   LIN {X -3.618, Y 42.239, Z 30.600} C_DIS
   LIN {X -4.278, Y 41.274, Z 30.600} C_DIS
   LIN {X -4.651, Y 40.757, Z 30.600} C_DIS
   LIN {X -4.747, Y 40.345, Z 30.600} C_DIS
   LIN {X -4.925, Y 39.487, Z 30.600} C_DIS
   LIN {X -4.816, Y 38.644, Z 30.600} C_DIS
   LIN {X -4.756, Y 38.144, Z 30.600} C_DIS
   LIN {X -4.582, Y 37.523, Z 30.600} C_DIS
   LIN {X -4.417, Y 36.940, Z 30.600} C_DIS
   LIN {X -4.292, Y 36.475, Z 30.600} C_DIS
   LIN {X -4.004, Y 35.393, Z 30.600} C_DIS
   LIN {X -3.515, Y 33.337, Z 30.600} C_DIS
   LIN {X -3.455, Y 33.086, Z 30.600} C_DIS
   LIN {X -3.401, Y 32.820, Z 30.600} C_DIS
   LIN {X -2.886, Y 30.247, Z 30.600} C_DIS
   LIN {X -2.481, Y 27.620, Z 30.600} C_DIS
   LIN {X -2.317, Y 26.540, Z 30.600} C_DIS
   LIN {X -2.260, Y 25.886, Z 30.600} C_DIS
   LIN {X -1.842, Y 21.391, Z 30.600} C_DIS
   LIN {X -1.832, Y 19.498, Z 30.600} C_DIS
   LIN {X -1.874, Y 12.631, Z 30.600} C_DIS
   LIN {X -2.420, Y 7.896, Z 30.600} C_DIS
   LIN {X -2.629, Y 5.941, Z 30.600} C_DIS
   LIN {X -2.726, Y 5.309, Z 30.600} C_DIS
   LIN {X -3.850, Y 0.233, Z 30.600} C_DIS
   LIN {X -4.314, Y -1.891, Z 30.600} C_DIS
   LIN {X -4.758, Y -3.318, Z 30.600} C_DIS
   LIN {X -5.741, Y -6.496, Z 30.600} C_DIS
   LIN {X -6.964, Y -9.707, Z 30.600} C_DIS
   LIN {X -7.355, Y -10.723, Z 30.600} C_DIS
   LIN {X -7.726, Y -11.533, Z 30.600} C_DIS
   LIN {X -9.075, Y -14.528, Z 30.600} C_DIS
   LIN {X -10.538, Y -17.348, Z 30.600} C_DIS
   LIN {X -10.853, Y -17.945, Z 30.600} C_DIS
   LIN {X -11.124, Y -18.727, Z 30.600} C_DIS
   LIN {X -11.882, Y -20.944, Z 30.600} C_DIS
   LIN {X -11.789, Y -22.564, Z 30.600} C_DIS
   LIN {X -11.686, Y -24.649, Z 30.600} C_DIS
   LIN {X -10.821, Y -26.557, Z 30.600} C_DIS
   LIN {X -10.384, Y -27.445, Z 30.600} C_DIS
   LIN {X -8.989, Y -28.695, Z 30.600} C_DIS
   LIN {X -7.458, Y -30.118, Z 30.600} C_DIS
   LIN {X -6.898, Y -30.342, Z 30.600} C_DIS
   LIN {X -4.652, Y -31.135, Z 30.600} C_DIS
   LIN {X -2.453, Y -31.231, Z 30.600} C_DIS
   LIN {X -2.161, Y -31.241, Z 30.600} C_DIS
   LIN {X -1.901, Y -31.152, Z 30.600}
   LaserEnd_Ext()
   LIN {X -6.660, Y -29.360, Z 30.600}
   LaserStart_Ext()
   LIN {X 0.314, Y -29.360, Z 30.600}
   LaserEnd_Ext()
   LIN {X 1.927, Y -28.360, Z 30.600}
   LaserStart_Ext()
   LIN {X -7.880, Y -28.360, Z 30.600}
   LaserEnd_Ext()
   LIN {X -8.980, Y -27.360, Z 30.600}
   LaserStart_Ext()
   LIN {X -6.021, Y -27.360, Z 30.600}
   LaserEnd_Ext()
   LIN {X 0.049, Y -27.360, Z 30.600}
   LaserStart_Ext()
   LIN {X 2.964, Y -27.360, Z 30.600}
   LaserEnd_Ext()
   LIN {X 3.806, Y -26.360, Z 30.600}
   LaserStart_Ext()
   LIN {X 1.372, Y -26.360, Z 30.600}
   LaserEnd_Ext()
   LIN {X -7.389, Y -26.360, Z 30.600}
   LaserStart_Ext()
   LIN {X -9.804, Y -26.360, Z 30.600}
   LaserEnd_Ext()
   LIN {X -10.266, Y -25.360, Z 30.600}
   LaserStart_Ext()
   LIN {X -8.010, Y -25.360, Z 30.600}
   LaserEnd_Ext()
   LIN {X 2.006, Y -25.360, Z 30.600}
   LaserStart_Ext()
   LIN {X 4.260, Y -25.360, Z 30.600}
   LaserEnd_Ext()
   LIN {X 4.715, Y -24.360, Z 30.600}
   LaserStart_Ext()
   LIN {X 2.517, Y -24.360, Z 30.600}
   LaserEnd_Ext()
   LIN {X -8.601, Y -24.360, Z 30.600}
   LaserStart_Ext()
   LIN {X -10.699, Y -24.360, Z 30.600}
   LaserEnd_Ext()
   LIN {X -10.748, Y -23.360, Z 30.600}
   LaserStart_Ext()
   LIN {X -8.789, Y -23.360, Z 30.600}
   LaserEnd_Ext()
   LIN {X 2.910, Y -23.360, Z 30.600}
   LaserStart_Ext()
   LIN {X 4.998, Y -23.360, Z 30.600}
   LaserEnd_Ext()
   LIN {X 5.242, Y -22.360, Z 30.600}
   LaserStart_Ext()
   LIN {X 2.915, Y -22.360, Z 30.600}
   LaserEnd_Ext()
   LIN {X -8.897, Y -22.360, Z 30.600}
   LaserStart_Ext()
   LIN {X -10.799, Y -22.360, Z 30.600}
   LaserEnd_Ext()
   LIN {X -10.856, Y -21.360, Z 30.600}
   LaserStart_Ext()
   LIN {X -8.848, Y -21.360, Z 30.600}
   LaserEnd_Ext()
   LIN {X 2.920, Y -21.360, Z 30.600}
   LaserStart_Ext()
   LIN {X 5.487, Y -21.360, Z 30.600}
   LaserEnd_Ext()
   LIN {X 5.712, Y -20.360, Z 30.600}
   LaserStart_Ext()
   LIN {X 2.625, Y -20.360, Z 30.600}
   LaserEnd_Ext()
   LIN {X -8.405, Y -20.360, Z 30.600}
   LaserStart_Ext()
   LIN {X -10.626, Y -20.360, Z 30.600}
   LaserEnd_Ext()
   LIN {X -10.284, Y -19.360, Z 30.600}
   LaserStart_Ext()
   LIN {X -7.968, Y -19.360, Z 30.600}
   LaserEnd_Ext()
   LIN {X 2.112, Y -19.360, Z 30.600}
   LaserStart_Ext()
   LIN {X 5.927, Y -19.360, Z 30.600}
   LaserEnd_Ext()
   LIN {X 6.139, Y -18.360, Z 30.600}
   LaserStart_Ext()
   LIN {X 1.590, Y -18.360, Z 30.600}
   LaserEnd_Ext()
   LIN {X -7.498, Y -18.360, Z 30.600}
   LaserStart_Ext()
   LIN {X -9.938, Y -18.360, Z 30.600}
   LaserEnd_Ext()
   LIN {X -9.418, Y -17.360, Z 30.600}
   LaserStart_Ext()
   LIN {X -6.233, Y -17.360, Z 30.600}
   LaserEnd_Ext()
   LIN {X 0.313, Y -17.360, Z 30.600}
   LaserStart_Ext()
   LIN {X 6.327, Y -17.360, Z 30.600}
   LaserEnd_Ext()
   LIN {X 6.509, Y -16.360, Z 30.600}
   LaserStart_Ext()
   LIN {X -2.524, Y -16.360, Z 30.600}
   LaserEnd_Ext()
   LIN {X -3.563, Y -16.360, Z 30.600}
   LaserStart_Ext()
   LIN {X -8.899, Y -16.360, Z 30.600}
   LaserEnd_Ext()
   LIN {X -8.380, Y -15.360, Z 30.600}
   LaserStart_Ext()
   LIN {X 6.691, Y -15.360, Z 30.600}
   LaserEnd_Ext()
   LIN {X 6.872, Y -14.360, Z 30.600}
   LaserStart_Ext()
   LIN {X -7.902, Y -14.360, Z 30.600}
   LaserEnd_Ext()
   LIN {X -7.452, Y -13.360, Z 30.600}
   LaserStart_Ext()
   LIN {X 7.014, Y -13.360, Z 30.600}
   LaserEnd_Ext()
   LIN {X 7.155, Y -12.360, Z 30.600}
   LaserStart_Ext()
   LIN {X -7.001, Y -12.360, Z 30.600}
   LaserEnd_Ext()
   LIN {X -6.547, Y -11.360, Z 30.600}
   LaserStart_Ext()
   LIN {X 7.297, Y -11.360, Z 30.600}
   LaserEnd_Ext()
   LIN {X 7.438, Y -10.360, Z 30.600}
   LaserStart_Ext()
   LIN {X -6.143, Y -10.360, Z 30.600}
   LaserEnd_Ext()
   LIN {X -5.761, Y -9.360, Z 30.600}
   LaserStart_Ext()
   LIN {X 7.568, Y -9.360, Z 30.600}
   LaserEnd_Ext()
   LIN {X 7.662, Y -8.360, Z 30.600}
   LaserStart_Ext()
   LIN {X -5.381, Y -8.360, Z 30.600}
   LaserEnd_Ext()
   LIN {X -5.000, Y -7.360, Z 30.600}
   LaserStart_Ext()
   LIN {X 7.756, Y -7.360, Z 30.600}
   LaserEnd_Ext()
   LIN {X 7.850, Y -6.360, Z 30.600}
   LaserStart_Ext()
   LIN {X -4.652, Y -6.360, Z 30.600}
   LaserEnd_Ext()
   LIN {X -4.343, Y -5.360, Z 30.600}
   LaserStart_Ext()
   LIN {X 7.941, Y -5.360, Z 30.600}
   LaserEnd_Ext()
   LIN {X 8.031, Y -4.360, Z 30.600}
   LaserStart_Ext()
   LIN {X -4.033, Y -4.360, Z 30.600}
   LaserEnd_Ext()
   LIN {X -3.723, Y -3.360, Z 30.600}
   LaserStart_Ext()
   LIN {X 8.100, Y -3.360, Z 30.600}
   LaserEnd_Ext()
   LIN {X 8.152, Y -2.360, Z 30.600}
   LaserStart_Ext()
   LIN {X -3.412, Y -2.360, Z 30.600}
   LaserEnd_Ext()
   LIN {X -3.174, Y -1.360, Z 30.600}
   LaserStart_Ext()
   LIN {X 8.186, Y -1.360, Z 30.600}
   LaserEnd_Ext()
   LIN {X 8.211, Y -0.360, Z 30.600}
   LaserStart_Ext()
   LIN {X -2.956, Y -0.360, Z 30.600}
   LaserEnd_Ext()
   LIN {X -2.735, Y 0.640, Z 30.600}
   LaserStart_Ext()
   LIN {X 8.237, Y 0.640, Z 30.600}
   LaserEnd_Ext()
   LIN {X 8.262, Y 1.640, Z 30.600}
   LaserStart_Ext()
   LIN {X -2.514, Y 1.640, Z 30.600}
   LaserEnd_Ext()
   LIN {X -2.293, Y 2.640, Z 30.600}
   LaserStart_Ext()
   LIN {X 8.288, Y 2.640, Z 30.600}
   LaserEnd_Ext()
   LIN {X 8.271, Y 3.640, Z 30.600}
   LaserStart_Ext()
   LIN {X -2.071, Y 3.640, Z 30.600}
   LaserEnd_Ext()
   LIN {X -1.850, Y 4.640, Z 30.600}
   LaserStart_Ext()
   LIN {X 8.247, Y 4.640, Z 30.600}
   LaserEnd_Ext()
   LIN {X 8.223, Y 5.640, Z 30.600}
   LaserStart_Ext()
   LIN {X -1.664, Y 5.640, Z 30.600}
   LaserEnd_Ext()
   LIN {X -1.549, Y 6.640, Z 30.600}
   LaserStart_Ext()
   LIN {X 8.199, Y 6.640, Z 30.600}
   LaserEnd_Ext()
   LIN {X 8.175, Y 7.640, Z 30.600}
   LaserStart_Ext()
   LIN {X -1.441, Y 7.640, Z 30.600}
   LaserEnd_Ext()
   LIN {X -1.327, Y 8.640, Z 30.600}
   LaserStart_Ext()
   LIN {X 8.137, Y 8.640, Z 30.600}
   LaserEnd_Ext()
   LIN {X 8.089, Y 9.640, Z 30.600}
   LaserStart_Ext()
   LIN {X -1.212, Y 9.640, Z 30.600}
   LaserEnd_Ext()
   LIN {X -1.097, Y 10.640, Z 30.600}
   LaserStart_Ext()
   LIN {X 8.042, Y 10.640, Z 30.600}
   LaserEnd_Ext()
   LIN {X 7.995, Y 11.640, Z 30.600}
   LaserStart_Ext()
   LIN {X -0.982, Y 11.640, Z 30.600}
   LaserEnd_Ext()
   LIN {X -0.874, Y 12.640, Z 30.600}
   LaserStart_Ext()
   LIN {X 7.910, Y 12.640, Z 30.600}
   LaserEnd_Ext()
   LIN {X 7.806, Y 13.640, Z 30.600}
   LaserStart_Ext()
   LIN {X -0.868, Y 13.640, Z 30.600}
   LaserEnd_Ext()
   LIN {X -0.862, Y 14.640, Z 30.600}
   LaserStart_Ext()
   LIN {X 7.702, Y 14.640, Z 30.600}
   LaserEnd_Ext()
   LIN {X 7.569, Y 15.640, Z 30.600}
   LaserStart_Ext()
   LIN {X -0.856, Y 15.640, Z 30.600}
   LaserEnd_Ext()
   LIN {X -0.850, Y 16.640, Z 30.600}
   LaserStart_Ext()
   LIN {X 7.431, Y 16.640, Z 30.600}
   LaserEnd_Ext()
   LIN {X 7.292, Y 17.640, Z 30.600}
   LaserStart_Ext()
   LIN {X -0.844, Y 17.640, Z 30.600}
   LaserEnd_Ext()
   LIN {X -0.838, Y 18.640, Z 30.600}
   LaserStart_Ext()
   LIN {X 7.154, Y 18.640, Z 30.600}
   LaserEnd_Ext()
   LIN {X 7.015, Y 19.640, Z 30.600}
   LaserStart_Ext()
   LIN {X -0.833, Y 19.640, Z 30.600}
   LaserEnd_Ext()
   LIN {X -0.838, Y 20.640, Z 30.600}
   LaserStart_Ext()
   LIN {X 6.864, Y 20.640, Z 30.600}
   LaserEnd_Ext()
   LIN {X 6.713, Y 21.640, Z 30.600}
   LaserStart_Ext()
   LIN {X -0.861, Y 21.640, Z 30.600}
   LaserEnd_Ext()
   LIN {X -0.954, Y 22.640, Z 30.600}
   LaserStart_Ext()
   LIN {X 6.561, Y 22.640, Z 30.600}
   LaserEnd_Ext()
   LIN {X 6.391, Y 23.640, Z 30.600}
   LaserStart_Ext()
   LIN {X -1.047, Y 23.640, Z 30.600}
   LaserEnd_Ext()
   LIN {X -1.139, Y 24.640, Z 30.600}
   LaserStart_Ext()
   LIN {X 6.173, Y 24.640, Z 30.600}
   LaserEnd_Ext()
   LIN {X 5.937, Y 25.640, Z 30.600}
   LaserStart_Ext()
   LIN {X -1.232, Y 25.640, Z 30.600}
   LaserEnd_Ext()
   LIN {X -1.323, Y 26.640, Z 30.600}
   LaserStart_Ext()
   LIN {X 5.697, Y 26.640, Z 30.600}
   LaserEnd_Ext()
   LIN {X 5.476, Y 27.640, Z 30.600}
   LaserStart_Ext()
   LIN {X -1.473, Y 27.640, Z 30.600}
   LaserEnd_Ext()
   LIN {X -1.627, Y 28.640, Z 30.600}
   LaserStart_Ext()
   LIN {X 5.270, Y 28.640, Z 30.600}
   LaserEnd_Ext()
   LIN {X 5.064, Y 29.640, Z 30.600}
   LaserStart_Ext()
   LIN {X -1.781, Y 29.640, Z 30.600}
   LaserEnd_Ext()
   LIN {X -1.945, Y 30.640, Z 30.600}
   LaserStart_Ext()
   LIN {X 4.824, Y 30.640, Z 30.600}
   LaserEnd_Ext()
   LIN {X 4.555, Y 31.640, Z 30.600}
   LaserStart_Ext()
   LIN {X -2.145, Y 31.640, Z 30.600}
   LaserEnd_Ext()
   LIN {X -2.345, Y 32.640, Z 30.600}
   LaserStart_Ext()
   LIN {X 4.287, Y 32.640, Z 30.600}
   LaserEnd_Ext()
   LIN {X 4.007, Y 33.640, Z 30.600}
   LaserStart_Ext()
   LIN {X -2.559, Y 33.640, Z 30.600}
   LaserEnd_Ext()
   LIN {X -2.797, Y 34.640, Z 30.600}
   LaserStart_Ext()
   LIN {X 3.712, Y 34.640, Z 30.600}
   LaserEnd_Ext()
   LIN {X 3.413, Y 35.640, Z 30.600}
   LaserStart_Ext()
   LIN {X -3.035, Y 35.640, Z 30.600}
   LaserEnd_Ext()
   LIN {X -3.301, Y 36.640, Z 30.600}
   LaserStart_Ext()
   LIN {X 3.097, Y 36.640, Z 30.600}
   LaserEnd_Ext()
   LIN {X 2.773, Y 37.640, Z 30.600}
   LaserStart_Ext()
   LIN {X -3.576, Y 37.640, Z 30.600}
   LaserEnd_Ext()
   LIN {X -3.808, Y 38.640, Z 30.600}
   LaserStart_Ext()
   LIN {X 2.438, Y 38.640, Z 30.600}
   LaserEnd_Ext()
   LIN {X 2.090, Y 39.640, Z 30.600}
   LaserStart_Ext()
   LIN {X -3.872, Y 39.640, Z 30.600}
   LaserEnd_Ext()
   LIN {X -3.502, Y 40.640, Z 30.600}
   LaserStart_Ext()
   LIN {X 1.632, Y 40.640, Z 30.600}
   LaserEnd_Ext()
   LIN {X 0.709, Y 41.640, Z 30.600}
   LaserStart_Ext()
   LIN {X -2.425, Y 41.640, Z 30.600}
   LaserEnd_Ext()
   LIN {X -5.717, Y -18.241, Z 31.450}
   LaserStart_Ext()
   LIN {X -5.008, Y -17.700, Z 31.450} C_DIS
   LIN {X -3.784, Y -17.409, Z 31.450} C_DIS
   LIN {X -3.008, Y -17.226, Z 31.450} C_DIS
   LIN {X -2.409, Y -17.339, Z 31.450} C_DIS
   LIN {X -0.901, Y -17.619, Z 31.450} C_DIS
   LIN {X 0.539, Y -18.651, Z 31.450} C_DIS
   LIN {X 0.826, Y -18.857, Z 31.450} C_DIS
   LIN {X 1.021, Y -19.237, Z 31.450} C_DIS
   LIN {X 1.994, Y -21.116, Z 31.450} C_DIS
   LIN {X 1.991, Y -22.729, Z 31.450} C_DIS
   LIN {X 1.988, Y -23.292, Z 31.450} C_DIS
   LIN {X 1.755, Y -23.747, Z 31.450} C_DIS
   LIN {X 0.880, Y -25.483, Z 31.450} C_DIS
   LIN {X -0.658, Y -26.657, Z 31.450} C_DIS
   LIN {X -0.782, Y -26.750, Z 31.450} C_DIS
   LIN {X -1.016, Y -26.803, Z 31.450} C_DIS
   LIN {X -2.872, Y -27.227, Z 31.450} C_DIS
   LIN {X -4.055, Y -26.995, Z 31.450} C_DIS
   LIN {X -4.899, Y -26.827, Z 31.450} C_DIS
   LIN {X -5.838, Y -26.159, Z 31.450} C_DIS
   LIN {X -6.583, Y -25.632, Z 31.450} C_DIS
   LIN {X -6.989, Y -24.951, Z 31.450} C_DIS
   LIN {X -7.647, Y -23.841, Z 31.450} C_DIS
   LIN {X -7.782, Y -22.606, Z 31.450} C_DIS
   LIN {X -7.876, Y -21.767, Z 31.450} C_DIS
   LIN {X -7.421, Y -20.706, Z 31.450} C_DIS
   LIN {X -6.650, Y -18.943, Z 31.450} C_DIS
   LIN {X -5.717, Y -18.241, Z 31.450}
   LaserEnd_Ext()
   LIN {X -7.202, Y -30.145, Z 31.450}
   LaserStart_Ext()
   LIN {X -7.333, Y -30.100, Z 31.450} C_DIS
   LIN {X -7.451, Y -30.002, Z 31.450} C_DIS
   LIN {X -10.203, Y -27.537, Z 31.450} C_DIS
   LIN {X -11.201, Y -25.513, Z 31.450} C_DIS
   LIN {X -11.604, Y -24.623, Z 31.450} C_DIS
   LIN {X -11.652, Y -23.650, Z 31.450} C_DIS
   LIN {X -11.809, Y -20.918, Z 31.450} C_DIS
   LIN {X -10.940, Y -18.374, Z 31.450} C_DIS
   LIN {X -10.787, Y -17.916, Z 31.450} C_DIS
   LIN {X -10.416, Y -17.192, Z 31.450} C_DIS
   LIN {X -9.022, Y -14.506, Z 31.450} C_DIS
   LIN {X -7.603, Y -11.355, Z 31.450} C_DIS
   LIN {X -7.335, Y -10.755, Z 31.450} C_DIS
   LIN {X -7.135, Y -10.224, Z 31.450} C_DIS
   LIN {X -5.720, Y -6.507, Z 31.450} C_DIS
   LIN {X -4.429, Y -2.333, Z 31.450} C_DIS
   LIN {X -4.342, Y -2.051, Z 31.450} C_DIS
   LIN {X -4.236, Y -1.572, Z 31.450} C_DIS
   LIN {X -2.754, Y 5.125, Z 31.450} C_DIS
   LIN {X -2.686, Y 5.572, Z 31.450} C_DIS
   LIN {X -2.537, Y 6.955, Z 31.450} C_DIS
   LIN {X -1.884, Y 12.627, Z 31.450} C_DIS
   LIN {X -1.848, Y 18.597, Z 31.450} C_DIS
   LIN {X -1.861, Y 21.319, Z 31.450} C_DIS
   LIN {X -2.299, Y 26.031, Z 31.450} C_DIS
   LIN {X -2.356, Y 26.579, Z 31.450} C_DIS
   LIN {X -2.912, Y 30.155, Z 31.450} C_DIS
   LIN {X -2.934, Y 30.294, Z 31.450} C_DIS
   LIN {X -2.965, Y 30.445, Z 31.450} C_DIS
   LIN {X -3.510, Y 33.132, Z 31.450} C_DIS
   LIN {X -3.950, Y 34.966, Z 31.450} C_DIS
   LIN {X -4.064, Y 35.438, Z 31.450} C_DIS
   LIN {X -4.163, Y 35.801, Z 31.450} C_DIS
   LIN {X -4.481, Y 36.983, Z 31.450} C_DIS
   LIN {X -4.646, Y 37.568, Z 31.450} C_DIS
   LIN {X -4.822, Y 38.187, Z 31.450} C_DIS
   LIN {X -4.952, Y 39.128, Z 31.450} C_DIS
   LIN {X -4.997, Y 39.480, Z 31.450} C_DIS
   LIN {X -4.933, Y 39.787, Z 31.450} C_DIS
   LIN {X -4.730, Y 40.786, Z 31.450} C_DIS
   LIN {X -3.916, Y 42.007, Z 31.450} C_DIS
   LIN {X -3.783, Y 42.202, Z 31.450} C_DIS
   LIN {X -3.444, Y 42.338, Z 31.450} C_DIS
   LIN {X -1.107, Y 43.314, Z 31.450} C_DIS
   LIN {X -0.169, Y 43.123, Z 31.450} C_DIS
   LIN {X 0.604, Y 42.964, Z 31.450} C_DIS
   LIN {X 1.747, Y 42.113, Z 31.450} C_DIS
   LIN {X 2.000, Y 41.925, Z 31.450} C_DIS
   LIN {X 2.087, Y 41.778, Z 31.450} C_DIS
   LIN {X 2.744, Y 40.655, Z 31.450} C_DIS
   LIN {X 3.191, Y 39.389, Z 31.450} C_DIS
   LIN {X 3.246, Y 39.232, Z 31.450} C_DIS
   LIN {X 3.477, Y 38.542, Z 31.450} C_DIS
   LIN {X 3.893, Y 37.300, Z 31.450} C_DIS
   LIN {X 4.023, Y 36.889, Z 31.450} C_DIS
   LIN {X 4.480, Y 35.439, Z 31.450} C_DIS
   LIN {X 4.741, Y 34.561, Z 31.450} C_DIS
   LIN {X 5.244, Y 32.823, Z 31.450} C_DIS
   LIN {X 5.775, Y 30.842, Z 31.450} C_DIS
   LIN {X 6.172, Y 28.912, Z 31.450} C_DIS
   LIN {X 6.972, Y 25.578, Z 31.450} C_DIS
   LIN {X 7.445, Y 23.404, Z 31.450} C_DIS
   LIN {X 8.277, Y 17.909, Z 31.450} C_DIS
   LIN {X 8.637, Y 15.308, Z 31.450} C_DIS
   LIN {X 8.987, Y 11.946, Z 31.450} C_DIS
   LIN {X 9.209, Y 7.250, Z 31.450} C_DIS
   LIN {X 9.310, Y 3.065, Z 31.450} C_DIS
   LIN {X 9.164, Y -2.691, Z 31.450} C_DIS
   LIN {X 9.094, Y -4.040, Z 31.450} C_DIS
   LIN {X 8.728, Y -8.094, Z 31.450} C_DIS
   LIN {X 8.571, Y -9.762, Z 31.450} C_DIS
   LIN {X 8.269, Y -11.897, Z 31.450} C_DIS
   LIN {X 7.918, Y -14.449, Z 31.450} C_DIS
   LIN {X 7.636, Y -16.049, Z 31.450} C_DIS
   LIN {X 7.235, Y -18.253, Z 31.450} C_DIS
   LIN {X 6.652, Y -21.011, Z 31.450} C_DIS
   LIN {X 6.600, Y -21.250, Z 31.450} C_DIS
   LIN {X 6.472, Y -21.773, Z 31.450} C_DIS
   LIN {X 5.835, Y -24.421, Z 31.450} C_DIS
   LIN {X 5.233, Y -25.767, Z 31.450} C_DIS
   LIN {X 4.574, Y -27.217, Z 31.450} C_DIS
   LIN {X 2.371, Y -29.339, Z 31.450} C_DIS
   LIN {X 1.831, Y -29.865, Z 31.450} C_DIS
   LIN {X 1.421, Y -30.017, Z 31.450} C_DIS
   LIN {X -1.962, Y -31.179, Z 31.450} C_DIS
   LIN {X -3.938, Y -31.107, Z 31.450} C_DIS
   LIN {X -4.513, Y -31.100, Z 31.450} C_DIS
   LIN {X -7.202, Y -30.145, Z 31.450}
   LaserEnd_Ext()
   LIN {X 7.602, Y -9.387, Z 31.450}
   LaserStart_Ext()
   LIN {X 7.602, Y 15.492, Z 31.450}
   LaserEnd_Ext()
   LIN {X 6.602, Y 22.292, Z 31.450}
   LaserStart_Ext()
   LIN {X 6.602, Y -16.145, Z 31.450}
   LaserEnd_Ext()
   LIN {X 5.602, Y -21.121, Z 31.450}
   LaserStart_Ext()
   LIN {X 5.602, Y 27.002, Z 31.450}
   LaserEnd_Ext()
   LIN {X 4.602, Y 31.355, Z 31.450}
   LaserStart_Ext()
   LIN {X 4.602, Y -24.728, Z 31.450}
   LaserEnd_Ext()
   LIN {X 3.602, Y -26.765, Z 31.450}
   LaserStart_Ext()
   LIN {X 3.602, Y 34.884, Z 31.450}
   LaserEnd_Ext()
   LIN {X 2.602, Y 38.005, Z 31.450}
   LaserStart_Ext()
   LIN {X 2.602, Y -20.115, Z 31.450}
   LaserEnd_Ext()
   LIN {X 2.602, Y -24.289, Z 31.450}
   LaserStart_Ext()
   LIN {X 2.602, Y -27.729, Z 31.450}
   LaserEnd_Ext()
   LIN {X 1.602, Y -28.693, Z 31.450}
   LaserStart_Ext()
   LIN {X 1.602, Y -26.174, Z 31.450}
   LaserEnd_Ext()
   LIN {X 1.602, Y -18.228, Z 31.450}
   LaserStart_Ext()
   LIN {X 1.602, Y 40.626, Z 31.450}
   LaserEnd_Ext()
   LIN {X 0.602, Y 41.719, Z 31.450}
   LaserStart_Ext()
   LIN {X 0.602, Y -17.466, Z 31.450}
   LaserEnd_Ext()
   LIN {X 0.602, Y -26.953, Z 31.450}
   LaserStart_Ext()
   LIN {X 0.602, Y -29.241, Z 31.450}
   LaserEnd_Ext()
   LIN {X -0.398, Y -29.585, Z 31.450}
   LaserStart_Ext()
   LIN {X -0.398, Y -27.672, Z 31.450}
   LaserEnd_Ext()
   LIN {X -0.398, Y -16.756, Z 31.450}
   LaserStart_Ext()
   LIN {X -0.398, Y 42.150, Z 31.450}
   LaserEnd_Ext()
   LIN {X -1.398, Y 42.109, Z 31.450}
   LaserStart_Ext()
   LIN {X -1.398, Y 26.928, Z 31.450}
   LaserEnd_Ext()
   LIN {X -1.398, Y 8.105, Z 31.450}
   LaserStart_Ext()
   LIN {X -1.398, Y -16.510, Z 31.450}
   LaserEnd_Ext()
   LIN {X -1.398, Y -27.916, Z 31.450}
   LaserStart_Ext()
   LIN {X -1.398, Y -29.928, Z 31.450}
   LaserEnd_Ext()
   LIN {X -2.398, Y -30.163, Z 31.450}
   LaserStart_Ext()
   LIN {X -2.398, Y -28.144, Z 31.450}
   LaserEnd_Ext()
   LIN {X -2.398, Y -16.323, Z 31.450}
   LaserStart_Ext()
   LIN {X -2.398, Y 2.106, Z 31.450}
   LaserEnd_Ext()
   LIN {X -2.398, Y 32.682, Z 31.450}
   LaserStart_Ext()
   LIN {X -2.398, Y 41.691, Z 31.450}
   LaserEnd_Ext()
   LIN {X -3.398, Y 40.982, Z 31.450}
   LaserStart_Ext()
   LIN {X -3.398, Y 36.808, Z 31.450}
   LaserEnd_Ext()
   LIN {X -3.398, Y -2.383, Z 31.450}
   LaserStart_Ext()
   LIN {X -3.398, Y -16.290, Z 31.450}
   LaserEnd_Ext()
   LIN {X -3.398, Y -28.143, Z 31.450}
   LaserStart_Ext()
   LIN {X -3.398, Y -30.126, Z 31.450}
   LaserEnd_Ext()
   LIN {X -4.398, Y -30.080, Z 31.450}
   LaserStart_Ext()
   LIN {X -4.398, Y -27.946, Z 31.450}
   LaserEnd_Ext()
   LIN {X -4.398, Y -16.527, Z 31.450}
   LaserStart_Ext()
   LIN {X -4.398, Y -5.618, Z 31.450}
   LaserEnd_Ext()
   LIN {X -5.398, Y -8.472, Z 31.450}
   LaserStart_Ext()
   LIN {X -5.398, Y -16.781, Z 31.450}
   LaserEnd_Ext()
   LIN {X -5.398, Y -27.694, Z 31.450}
   LaserStart_Ext()
   LIN {X -5.398, Y -29.724, Z 31.450}
   LaserEnd_Ext()
   LIN {X -6.398, Y -29.369, Z 31.450}
   LaserStart_Ext()
   LIN {X -6.398, Y -26.988, Z 31.450}
   LaserEnd_Ext()
   LIN {X -6.398, Y -17.502, Z 31.450}
   LaserStart_Ext()
   LIN {X -6.398, Y -11.105, Z 31.450}
   LaserEnd_Ext()
   LIN {X -7.398, Y -13.335, Z 31.450}
   LaserStart_Ext()
   LIN {X -7.398, Y -18.280, Z 31.450}
   LaserEnd_Ext()
   LIN {X -7.398, Y -26.209, Z 31.450}
   LaserStart_Ext()
   LIN {X -7.398, Y -28.707, Z 31.450}
   LaserEnd_Ext()
   LIN {X -8.398, Y -27.811, Z 31.450}
   LaserStart_Ext()
   LIN {X -8.398, Y -24.536, Z 31.450}
   LaserEnd_Ext()
   LIN {X -8.398, Y -20.448, Z 31.450}
   LaserStart_Ext()
   LIN {X -8.398, Y -15.474, Z 31.450}
   LaserEnd_Ext()
   LIN {X -9.398, Y -17.401, Z 31.450}
   LaserStart_Ext()
   LIN {X -9.398, Y -26.909, Z 31.450}
   LaserEnd_Ext()
   LIN {X -10.398, Y -24.862, Z 31.450}
   LaserStart_Ext()
   LIN {X -10.398, Y -19.882, Z 31.450}
   LaserEnd_Ext()
   LIN {X -2.796, Y -27.179, Z 32.300}
   LaserStart_Ext()
   LIN {X -4.245, Y -26.895, Z 32.300} C_DIS
   LIN {X -4.813, Y -26.785, Z 32.300} C_DIS
   LIN {X -5.177, Y -26.529, Z 32.300} C_DIS
   LIN {X -6.499, Y -25.593, Z 32.300} C_DIS
   LIN {X -7.463, Y -23.980, Z 32.300} C_DIS
   LIN {X -7.568, Y -23.805, Z 32.300} C_DIS
   LIN {X -7.590, Y -23.612, Z 32.300} C_DIS
   LIN {X -7.802, Y -21.731, Z 32.300} C_DIS
   LIN {X -6.614, Y -18.964, Z 32.300} C_DIS
   LIN {X -4.937, Y -17.655, Z 32.300} C_DIS
   LIN {X -2.934, Y -17.178, Z 32.300} C_DIS
   LIN {X -2.093, Y -17.333, Z 32.300} C_DIS
   LIN {X -0.836, Y -17.567, Z 32.300} C_DIS
   LIN {X 0.042, Y -18.196, Z 32.300} C_DIS
   LIN {X 0.893, Y -18.800, Z 32.300} C_DIS
   LIN {X 1.517, Y -19.995, Z 32.300} C_DIS
   LIN {X 2.067, Y -21.057, Z 32.300} C_DIS
   LIN {X 2.065, Y -22.216, Z 32.300} C_DIS
   LIN {X 2.066, Y -23.233, Z 32.300} C_DIS
   LIN {X 1.275, Y -24.812, Z 32.300} C_DIS
   LIN {X 0.967, Y -25.422, Z 32.300} C_DIS
   LIN {X 0.622, Y -25.686, Z 32.300} C_DIS
   LIN {X -0.683, Y -26.691, Z 32.300} C_DIS
   LIN {X -1.785, Y -26.948, Z 32.300} C_DIS
   LIN {X -2.796, Y -27.179, Z 32.300}
   LaserEnd_Ext()
   LIN {X 4.664, Y -27.150, Z 32.300}
   LaserStart_Ext()
   LIN {X 4.229, Y -27.568, Z 32.300} C_DIS
   LIN {X 1.936, Y -29.800, Z 32.300} C_DIS
   LIN {X 0.194, Y -30.445, Z 32.300} C_DIS
   LIN {X -1.762, Y -31.117, Z 32.300} C_DIS
   LIN {X -2.905, Y -31.075, Z 32.300} C_DIS
   LIN {X -4.408, Y -31.057, Z 32.300} C_DIS
   LIN {X -6.317, Y -30.380, Z 32.300} C_DIS
   LIN {X -7.237, Y -30.063, Z 32.300} C_DIS
   LIN {X -8.072, Y -29.376, Z 32.300} C_DIS
   LIN {X -10.023, Y -27.629, Z 32.300} C_DIS
   LIN {X -11.437, Y -24.759, Z 32.300} C_DIS
   LIN {X -11.523, Y -24.596, Z 32.300} C_DIS
   LIN {X -11.538, Y -24.342, Z 32.300} C_DIS
   LIN {X -11.736, Y -20.891, Z 32.300} C_DIS
   LIN {X -11.188, Y -19.289, Z 32.300} C_DIS
   LIN {X -10.721, Y -17.888, Z 32.300} C_DIS
   LIN {X -9.586, Y -15.672, Z 32.300} C_DIS
   LIN {X -8.969, Y -14.483, Z 32.300} C_DIS
   LIN {X -8.341, Y -13.089, Z 32.300} C_DIS
   LIN {X -7.327, Y -10.818, Z 32.300} C_DIS
   LIN {X -6.572, Y -8.810, Z 32.300} C_DIS
   LIN {X -5.699, Y -6.518, Z 32.300} C_DIS
   LIN {X -4.903, Y -3.945, Z 32.300} C_DIS
   LIN {X -4.340, Y -2.108, Z 32.300} C_DIS
   LIN {X -3.652, Y 1.011, Z 32.300} C_DIS
   LIN {X -2.782, Y 4.941, Z 32.300} C_DIS
   LIN {X -2.742, Y 5.203, Z 32.300} C_DIS
   LIN {X -2.655, Y 6.015, Z 32.300} C_DIS
   LIN {X -1.893, Y 12.624, Z 32.300} C_DIS
   LIN {X -1.863, Y 17.695, Z 32.300} C_DIS
   LIN {X -1.880, Y 21.247, Z 32.300} C_DIS
   LIN {X -2.251, Y 25.238, Z 32.300} C_DIS
   LIN {X -2.395, Y 26.628, Z 32.300} C_DIS
   LIN {X -2.982, Y 30.341, Z 32.300} C_DIS
   LIN {X -3.375, Y 32.263, Z 32.300} C_DIS
   LIN {X -3.564, Y 33.178, Z 32.300} C_DIS
   LIN {X -3.746, Y 33.923, Z 32.300} C_DIS
   LIN {X -4.124, Y 35.483, Z 32.300} C_DIS
   LIN {X -4.376, Y 36.413, Z 32.300} C_DIS
   LIN {X -4.544, Y 37.027, Z 32.300} C_DIS
   LIN {X -4.739, Y 37.706, Z 32.300} C_DIS
   LIN {X -4.889, Y 38.230, Z 32.300} C_DIS
   LIN {X -4.940, Y 38.602, Z 32.300} C_DIS
   LIN {X -5.067, Y 39.511, Z 32.300} C_DIS
   LIN {X -4.820, Y 40.724, Z 32.300} C_DIS
   LIN {X -4.793, Y 40.854, Z 32.300} C_DIS
   LIN {X -4.713, Y 40.975, Z 32.300} C_DIS
   LIN {X -3.866, Y 42.240, Z 32.300} C_DIS
   LIN {X -3.583, Y 42.458, Z 32.300} C_DIS
   LIN {X -2.040, Y 43.009, Z 32.300} C_DIS
   LIN {X -1.185, Y 43.365, Z 32.300} C_DIS
   LIN {X -0.330, Y 43.192, Z 32.300} C_DIS
   LIN {X 0.526, Y 43.020, Z 32.300} C_DIS
   LIN {X 1.009, Y 42.664, Z 32.300} C_DIS
   LIN {X 1.925, Y 41.984, Z 32.300} C_DIS
   LIN {X 2.653, Y 40.747, Z 32.300} C_DIS
   LIN {X 3.169, Y 39.316, Z 32.300} C_DIS
   LIN {X 3.621, Y 37.984, Z 32.300} C_DIS
   LIN {X 3.795, Y 37.465, Z 32.300} C_DIS
   LIN {X 4.490, Y 35.270, Z 32.300} C_DIS
   LIN {X 4.547, Y 35.089, Z 32.300} C_DIS
   LIN {X 4.579, Y 34.979, Z 32.300} C_DIS
   LIN {X 5.364, Y 32.263, Z 32.300} C_DIS
   LIN {X 5.599, Y 31.386, Z 32.300} C_DIS
   LIN {X 5.776, Y 30.532, Z 32.300} C_DIS
   LIN {X 6.829, Y 26.137, Z 32.300} C_DIS
   LIN {X 7.453, Y 23.272, Z 32.300} C_DIS
   LIN {X 8.549, Y 16.032, Z 32.300} C_DIS
   LIN {X 8.597, Y 15.682, Z 32.300} C_DIS
   LIN {X 8.998, Y 11.830, Z 32.300} C_DIS
   LIN {X 9.253, Y 6.448, Z 32.300} C_DIS
   LIN {X 9.328, Y 3.336, Z 32.300} C_DIS
   LIN {X 9.158, Y -3.325, Z 32.300} C_DIS
   LIN {X 9.119, Y -4.081, Z 32.300} C_DIS
   LIN {X 8.658, Y -9.193, Z 32.300} C_DIS
   LIN {X 8.606, Y -9.786, Z 32.300} C_DIS
   LIN {X 8.571, Y -10.054, Z 32.300} C_DIS
   LIN {X 7.972, Y -14.398, Z 32.300} C_DIS
   LIN {X 7.422, Y -17.520, Z 32.300} C_DIS
   LIN {X 7.302, Y -18.182, Z 32.300} C_DIS
   LIN {X 7.076, Y -19.252, Z 32.300} C_DIS
   LIN {X 6.674, Y -21.180, Z 32.300} C_DIS
   LIN {X 6.462, Y -22.087, Z 32.300} C_DIS
   LIN {X 5.916, Y -24.353, Z 32.300} C_DIS
   LIN {X 4.793, Y -26.864, Z 32.300} C_DIS
   LIN {X 4.664, Y -27.150, Z 32.300}
   LaserEnd_Ext()
   LIN {X -3.144, Y 41.522, Z 32.300}
   LaserStart_Ext()
   LIN {X 0.870, Y 41.522, Z 32.300}
   LaserEnd_Ext()
   LIN {X 1.625, Y 40.522, Z 32.300}
   LaserStart_Ext()
   LIN {X -3.812, Y 40.522, Z 32.300}
   LaserEnd_Ext()
   LIN {X -4.044, Y 39.522, Z 32.300}
   LaserStart_Ext()
   LIN {X 2.035, Y 39.522, Z 32.300}
   LaserEnd_Ext()
   LIN {X 2.383, Y 38.522, Z 32.300}
   LaserStart_Ext()
   LIN {X -3.919, Y 38.522, Z 32.300}
   LaserEnd_Ext()
   LIN {X -3.646, Y 37.522, Z 32.300}
   LaserStart_Ext()
   LIN {X 2.722, Y 37.522, Z 32.300}
   LaserEnd_Ext()
   LIN {X 3.045, Y 36.522, Z 32.300}
   LaserStart_Ext()
   LIN {X -3.370, Y 36.522, Z 32.300}
   LaserEnd_Ext()
   LIN {X -3.105, Y 35.522, Z 32.300}
   LaserStart_Ext()
   LIN {X 3.361, Y 35.522, Z 32.300}
   LaserEnd_Ext()
   LIN {X 3.670, Y 34.522, Z 32.300}
   LaserStart_Ext()
   LIN {X -2.862, Y 34.522, Z 32.300}
   LaserEnd_Ext()
   LIN {X -2.619, Y 33.522, Z 32.300}
   LaserStart_Ext()
   LIN {X 3.959, Y 33.522, Z 32.300}
   LaserEnd_Ext()
   LIN {X 4.249, Y 32.522, Z 32.300}
   LaserStart_Ext()
   LIN {X -2.407, Y 32.522, Z 32.300}
   LaserEnd_Ext()
   LIN {X -2.203, Y 31.522, Z 32.300}
   LaserStart_Ext()
   LIN {X 4.528, Y 31.522, Z 32.300}
   LaserEnd_Ext()
   LIN {X 4.757, Y 30.522, Z 32.300}
   LaserStart_Ext()
   LIN {X -1.999, Y 30.522, Z 32.300}
   LaserEnd_Ext()
   LIN {X -1.840, Y 29.522, Z 32.300}
   LaserStart_Ext()
   LIN {X 4.989, Y 29.522, Z 32.300}
   LaserEnd_Ext()
   LIN {X 5.229, Y 28.522, Z 32.300}
   LaserStart_Ext()
   LIN {X -1.682, Y 28.522, Z 32.300}
   LaserEnd_Ext()
   LIN {X -1.524, Y 27.522, Z 32.300}
   LaserStart_Ext()
   LIN {X 5.469, Y 27.522, Z 32.300}
   LaserEnd_Ext()
   LIN {X 5.709, Y 26.522, Z 32.300}
   LaserStart_Ext()
   LIN {X -1.379, Y 26.522, Z 32.300}
   LaserEnd_Ext()
   LIN {X -1.275, Y 25.522, Z 32.300}
   LaserStart_Ext()
   LIN {X 5.940, Y 25.522, Z 32.300}
   LaserEnd_Ext()
   LIN {X 6.157, Y 24.522, Z 32.300}
   LaserStart_Ext()
   LIN {X -1.180, Y 24.522, Z 32.300}
   LaserEnd_Ext()
   LIN {X -1.087, Y 23.522, Z 32.300}
   LaserStart_Ext()
   LIN {X 6.375, Y 23.522, Z 32.300}
   LaserEnd_Ext()
   LIN {X 6.555, Y 22.522, Z 32.300}
   LaserStart_Ext()
   LIN {X -0.994, Y 22.522, Z 32.300}
   LaserEnd_Ext()
   LIN {X -0.901, Y 21.522, Z 32.300}
   LaserStart_Ext()
   LIN {X 6.707, Y 21.522, Z 32.300}
   LaserEnd_Ext()
   LIN {X 6.858, Y 20.522, Z 32.300}
   LaserStart_Ext()
   LIN {X -0.876, Y 20.522, Z 32.300}
   LaserEnd_Ext()
   LIN {X -0.872, Y 19.522, Z 32.300}
   LaserStart_Ext()
   LIN {X 7.009, Y 19.522, Z 32.300}
   LaserEnd_Ext()
   LIN {X 7.161, Y 18.522, Z 32.300}
   LaserStart_Ext()
   LIN {X -0.867, Y 18.522, Z 32.300}
   LaserEnd_Ext()
   LIN {X -0.864, Y 17.522, Z 32.300}
   LaserStart_Ext()
   LIN {X 7.312, Y 17.522, Z 32.300}
   LaserEnd_Ext()
   LIN {X 7.463, Y 16.522, Z 32.300}
   LaserStart_Ext()
   LIN {X -0.870, Y 16.522, Z 32.300}
   LaserEnd_Ext()
   LIN {X -0.876, Y 15.522, Z 32.300}
   LaserStart_Ext()
   LIN {X 7.608, Y 15.522, Z 32.300}
   LaserEnd_Ext()
   LIN {X 7.713, Y 14.522, Z 32.300}
   LaserStart_Ext()
   LIN {X -0.882, Y 14.522, Z 32.300}
   LaserEnd_Ext()
   LIN {X -0.888, Y 13.522, Z 32.300}
   LaserStart_Ext()
   LIN {X 7.817, Y 13.522, Z 32.300}
   LaserEnd_Ext()
   LIN {X 7.921, Y 12.522, Z 32.300}
   LaserStart_Ext()
   LIN {X -0.899, Y 12.522, Z 32.300}
   LaserEnd_Ext()
   LIN {X -1.014, Y 11.522, Z 32.300}
   LaserStart_Ext()
   LIN {X 8.012, Y 11.522, Z 32.300}
   LaserEnd_Ext()
   LIN {X 8.059, Y 10.522, Z 32.300}
   LaserStart_Ext()
   LIN {X -1.129, Y 10.522, Z 32.300}
   LaserEnd_Ext()
   LIN {X -1.244, Y 9.522, Z 32.300}
   LaserStart_Ext()
   LIN {X 8.106, Y 9.522, Z 32.300}
   LaserEnd_Ext()
   LIN {X 8.154, Y 8.522, Z 32.300}
   LaserStart_Ext()
   LIN {X -1.359, Y 8.522, Z 32.300}
   LaserEnd_Ext()
   LIN {X -1.474, Y 7.522, Z 32.300}
   LaserStart_Ext()
   LIN {X 8.201, Y 7.522, Z 32.300}
   LaserEnd_Ext()
   LIN {X 8.248, Y 6.522, Z 32.300}
   LaserStart_Ext()
   LIN {X -1.590, Y 6.522, Z 32.300}
   LaserEnd_Ext()
   LIN {X -1.702, Y 5.522, Z 32.300}
   LaserStart_Ext()
   LIN {X 8.275, Y 5.522, Z 32.300}
   LaserEnd_Ext()
   LIN {X 8.299, Y 4.522, Z 32.300}
   LaserStart_Ext()
   LIN {X -1.850, Y 4.522, Z 32.300}
   LaserEnd_Ext()
   LIN {X -2.072, Y 3.522, Z 32.300}
   LaserStart_Ext()
   LIN {X 8.323, Y 3.522, Z 32.300}
   LaserEnd_Ext()
   LIN {X 8.307, Y 2.522, Z 32.300}
   LaserStart_Ext()
   LIN {X -2.293, Y 2.522, Z 32.300}
   LaserEnd_Ext()
   LIN {X -2.515, Y 1.522, Z 32.300}
   LaserStart_Ext()
   LIN {X 8.281, Y 1.522, Z 32.300}
   LaserEnd_Ext()
   LIN {X 8.256, Y 0.522, Z 32.300}
   LaserStart_Ext()
   LIN {X -2.736, Y 0.522, Z 32.300}
   LaserEnd_Ext()
   LIN {X -2.956, Y -0.478, Z 32.300}
   LaserStart_Ext()
   LIN {X 8.230, Y -0.478, Z 32.300}
   LaserEnd_Ext()
   LIN {X 8.205, Y -1.478, Z 32.300}
   LaserStart_Ext()
   LIN {X -3.177, Y -1.478, Z 32.300}
   LaserEnd_Ext()
   LIN {X -3.408, Y -2.478, Z 32.300}
   LaserStart_Ext()
   LIN {X 8.180, Y -2.478, Z 32.300}
   LaserEnd_Ext()
   LIN {X 8.149, Y -3.478, Z 32.300}
   LaserStart_Ext()
   LIN {X -3.714, Y -3.478, Z 32.300}
   LaserEnd_Ext()
   LIN {X -4.021, Y -4.478, Z 32.300}
   LaserStart_Ext()
   LIN {X 8.079, Y -4.478, Z 32.300}
   LaserEnd_Ext()
   LIN {X 7.989, Y -5.478, Z 32.300}
   LaserStart_Ext()
   LIN {X -4.330, Y -5.478, Z 32.300}
   LaserEnd_Ext()
   LIN {X -4.640, Y -6.478, Z 32.300}
   LaserStart_Ext()
   LIN {X 7.899, Y -6.478, Z 32.300}
   LaserEnd_Ext()
   LIN {X 7.808, Y -7.478, Z 32.300}
   LaserStart_Ext()
   LIN {X -4.994, Y -7.478, Z 32.300}
   LaserEnd_Ext()
   LIN {X -5.375, Y -8.478, Z 32.300}
   LaserStart_Ext()
   LIN {X 7.718, Y -8.478, Z 32.300}
   LaserEnd_Ext()
   LIN {X 7.629, Y -9.478, Z 32.300}
   LaserStart_Ext()
   LIN {X -5.755, Y -9.478, Z 32.300}
   LaserEnd_Ext()
   LIN {X -6.130, Y -10.478, Z 32.300}
   LaserStart_Ext()
   LIN {X 7.503, Y -10.478, Z 32.300}
   LaserEnd_Ext()
   LIN {X 7.365, Y -11.478, Z 32.300}
   LaserStart_Ext()
   LIN {X -6.526, Y -11.478, Z 32.300}
   LaserEnd_Ext()
   LIN {X -6.973, Y -12.478, Z 32.300}
   LaserStart_Ext()
   LIN {X 7.227, Y -12.478, Z 32.300}
   LaserEnd_Ext()
   LIN {X 7.089, Y -13.478, Z 32.300}
   LaserStart_Ext()
   LIN {X -7.420, Y -13.478, Z 32.300}
   LaserEnd_Ext()
   LIN {X -7.870, Y -14.478, Z 32.300}
   LaserStart_Ext()
   LIN {X 6.942, Y -14.478, Z 32.300}
   LaserEnd_Ext()
   LIN {X 6.766, Y -15.478, Z 32.300}
   LaserStart_Ext()
   LIN {X -8.359, Y -15.478, Z 32.300}
   LaserEnd_Ext()
   LIN {X -8.876, Y -16.478, Z 32.300}
   LaserStart_Ext()
   LIN {X -4.312, Y -16.478, Z 32.300}
   LaserEnd_Ext()
   LIN {X -1.222, Y -16.478, Z 32.300}
   LaserStart_Ext()
   LIN {X 6.590, Y -16.478, Z 32.300}
   LaserEnd_Ext()
   LIN {X 6.414, Y -17.478, Z 32.300}
   LaserStart_Ext()
   LIN {X 0.759, Y -17.478, Z 32.300}
   LaserEnd_Ext()
   LIN {X -6.355, Y -17.478, Z 32.300}
   LaserStart_Ext()
   LIN {X -9.388, Y -17.478, Z 32.300}
   LaserEnd_Ext()
   LIN {X -9.864, Y -18.478, Z 32.300}
   LaserStart_Ext()
   LIN {X -7.491, Y -18.478, Z 32.300}
   LaserEnd_Ext()
   LIN {X 1.853, Y -18.478, Z 32.300}
   LaserStart_Ext()
   LIN {X 6.217, Y -18.478, Z 32.300}
   LaserEnd_Ext()
   LIN {X 6.007, Y -19.478, Z 32.300}
   LaserStart_Ext()
   LIN {X 2.375, Y -19.478, Z 32.300}
   LaserEnd_Ext()
   LIN {X -7.923, Y -19.478, Z 32.300}
   LaserStart_Ext()
   LIN {X -10.197, Y -19.478, Z 32.300}
   LaserEnd_Ext()
   LIN {X -10.538, Y -20.478, Z 32.300}
   LaserStart_Ext()
   LIN {X -8.352, Y -20.478, Z 32.300}
   LaserEnd_Ext()
   LIN {X 2.894, Y -20.478, Z 32.300}
   LaserStart_Ext()
   LIN {X 5.799, Y -20.478, Z 32.300}
   LaserEnd_Ext()
   LIN {X 5.577, Y -21.478, Z 32.300}
   LaserStart_Ext()
   LIN {X 3.066, Y -21.478, Z 32.300}
   LaserEnd_Ext()
   LIN {X -8.768, Y -21.478, Z 32.300}
   LaserStart_Ext()
   LIN {X -10.700, Y -21.478, Z 32.300}
   LaserEnd_Ext()
   LIN {X -10.643, Y -22.478, Z 32.300}
   LaserStart_Ext()
   LIN {X -8.724, Y -22.478, Z 32.300}
   LaserEnd_Ext()
   LIN {X 3.065, Y -22.478, Z 32.300}
   LaserStart_Ext()
   LIN {X 5.339, Y -22.478, Z 32.300}
   LaserEnd_Ext()
   LIN {X 5.098, Y -23.478, Z 32.300}
   LaserStart_Ext()
   LIN {X 3.035, Y -23.478, Z 32.300}
   LaserEnd_Ext()
   LIN {X -8.611, Y -23.478, Z 32.300}
   LaserStart_Ext()
   LIN {X -10.586, Y -23.478, Z 32.300}
   LaserEnd_Ext()
   LIN {X -10.461, Y -24.478, Z 32.300}
   LaserStart_Ext()
   LIN {X -8.330, Y -24.478, Z 32.300}
   LaserEnd_Ext()
   LIN {X 2.561, Y -24.478, Z 32.300}
   LaserStart_Ext()
   LIN {X 4.765, Y -24.478, Z 32.300}
   LaserEnd_Ext()
   LIN {X 4.318, Y -25.478, Z 32.300}
   LaserStart_Ext()
   LIN {X 2.059, Y -25.478, Z 32.300}
   LaserEnd_Ext()
   LIN {X -7.732, Y -25.478, Z 32.300}
   LaserStart_Ext()
   LIN {X -9.968, Y -25.478, Z 32.300}
   LaserEnd_Ext()
   LIN {X -9.475, Y -26.478, Z 32.300}
   LaserStart_Ext()
   LIN {X -6.979, Y -26.478, Z 32.300}
   LaserEnd_Ext()
   LIN {X 1.232, Y -26.478, Z 32.300}
   LaserStart_Ext()
   LIN {X 3.870, Y -26.478, Z 32.300}
   LaserEnd_Ext()
   LIN {X 2.888, Y -27.478, Z 32.300}
   LaserStart_Ext()
   LIN {X -0.067, Y -27.478, Z 32.300}
   LaserEnd_Ext()
   LIN {X -5.565, Y -27.478, Z 32.300}
   LaserStart_Ext()
   LIN {X -8.692, Y -27.478, Z 32.300}
   LaserEnd_Ext()
   LIN {X -7.576, Y -28.478, Z 32.300}
   LaserStart_Ext()
   LIN {X 1.860, Y -28.478, Z 32.300}
   LaserEnd_Ext()
   LIN {X -0.075, Y -29.478, Z 32.300}
   LaserStart_Ext()
   LIN {X -5.866, Y -29.478, Z 32.300}
   LaserEnd_Ext()
   LIN {X -4.667, Y -17.562, Z 33.150}
   LaserStart_Ext()
   LIN {X -2.857, Y -17.130, Z 33.150} C_DIS
   LIN {X -1.043, Y -17.465, Z 33.150} C_DIS
   LIN {X -0.772, Y -17.515, Z 33.150} C_DIS
   LIN {X -0.491, Y -17.713, Z 33.150} C_DIS
   LIN {X 0.961, Y -18.744, Z 33.150} C_DIS
   LIN {X 1.868, Y -20.480, Z 33.150} C_DIS
   LIN {X 2.140, Y -20.997, Z 33.150} C_DIS
   LIN {X 2.142, Y -21.444, Z 33.150} C_DIS
   LIN {X 2.145, Y -23.174, Z 33.150} C_DIS
   LIN {X 1.468, Y -24.524, Z 33.150} C_DIS
   LIN {X 1.054, Y -25.361, Z 33.150} C_DIS
   LIN {X 0.306, Y -25.947, Z 33.150} C_DIS
   LIN {X -0.583, Y -26.632, Z 33.150} C_DIS
   LIN {X -2.361, Y -27.047, Z 33.150} C_DIS
   LIN {X -2.717, Y -27.131, Z 33.150} C_DIS
   LIN {X -2.948, Y -27.087, Z 33.150} C_DIS
   LIN {X -4.726, Y -26.741, Z 33.150} C_DIS
   LIN {X -6.219, Y -25.693, Z 33.150} C_DIS
   LIN {X -6.416, Y -25.554, Z 33.150} C_DIS
   LIN {X -6.559, Y -25.313, Z 33.150} C_DIS
   LIN {X -7.488, Y -23.768, Z 33.150} C_DIS
   LIN {X -7.685, Y -22.070, Z 33.150} C_DIS
   LIN {X -7.727, Y -21.695, Z 33.150} C_DIS
   LIN {X -7.490, Y -21.144, Z 33.150} C_DIS
   LIN {X -6.536, Y -18.890, Z 33.150} C_DIS
   LIN {X -5.104, Y -17.790, Z 33.150} C_DIS
   LIN {X -4.867, Y -17.610, Z 33.150} C_DIS
   LIN {X -4.667, Y -17.562, Z 33.150}
   LaserEnd_Ext()
   LIN {X 9.153, Y -3.960, Z 33.150}
   LaserStart_Ext()
   LIN {X 9.145, Y -4.121, Z 33.150} C_DIS
   LIN {X 9.046, Y -5.214, Z 33.150} C_DIS
   LIN {X 8.653, Y -9.711, Z 33.150} C_DIS
   LIN {X 8.385, Y -11.744, Z 33.150} C_DIS
   LIN {X 8.026, Y -14.347, Z 33.150} C_DIS
   LIN {X 7.545, Y -17.079, Z 33.150} C_DIS
   LIN {X 7.367, Y -18.123, Z 33.150} C_DIS
   LIN {X 7.248, Y -18.710, Z 33.150} C_DIS
   LIN {X 6.748, Y -21.109, Z 33.150} C_DIS
   LIN {X 6.261, Y -23.193, Z 33.150} C_DIS
   LIN {X 5.998, Y -24.285, Z 33.150} C_DIS
   LIN {X 5.308, Y -25.829, Z 33.150} C_DIS
   LIN {X 4.758, Y -27.075, Z 33.150} C_DIS
   LIN {X 3.979, Y -27.848, Z 33.150} C_DIS
   LIN {X 2.040, Y -29.734, Z 33.150} C_DIS
   LIN {X -1.033, Y -30.873, Z 33.150} C_DIS
   LIN {X -1.563, Y -31.055, Z 33.150} C_DIS
   LIN {X -1.872, Y -31.044, Z 33.150} C_DIS
   LIN {X -4.304, Y -31.015, Z 33.150} C_DIS
   LIN {X -5.432, Y -30.614, Z 33.150} C_DIS
   LIN {X -7.142, Y -30.025, Z 33.150} C_DIS
   LIN {X -8.693, Y -28.750, Z 33.150} C_DIS
   LIN {X -9.842, Y -27.720, Z 33.150} C_DIS
   LIN {X -10.676, Y -26.030, Z 33.150} C_DIS
   LIN {X -11.441, Y -24.569, Z 33.150} C_DIS
   LIN {X -11.581, Y -22.290, Z 33.150} C_DIS
   LIN {X -11.663, Y -20.865, Z 33.150} C_DIS
   LIN {X -11.437, Y -20.204, Z 33.150} C_DIS
   LIN {X -10.655, Y -17.859, Z 33.150} C_DIS
   LIN {X -9.038, Y -14.702, Z 33.150} C_DIS
   LIN {X -8.921, Y -14.471, Z 33.150} C_DIS
   LIN {X -8.818, Y -14.237, Z 33.150} C_DIS
   LIN {X -7.319, Y -10.882, Z 33.150} C_DIS
   LIN {X -6.008, Y -7.396, Z 33.150} C_DIS
   LIN {X -5.678, Y -6.530, Z 33.150} C_DIS
   LIN {X -5.377, Y -5.557, Z 33.150} C_DIS
   LIN {X -4.338, Y -2.166, Z 33.150} C_DIS
   LIN {X -3.067, Y 3.594, Z 33.150} C_DIS
   LIN {X -2.810, Y 4.757, Z 33.150} C_DIS
   LIN {X -2.772, Y 5.075, Z 33.150} C_DIS
   LIN {X -1.903, Y 12.620, Z 33.150} C_DIS
   LIN {X -1.878, Y 16.793, Z 33.150} C_DIS
   LIN {X -1.899, Y 21.175, Z 33.150} C_DIS
   LIN {X -2.203, Y 24.445, Z 33.150} C_DIS
   LIN {X -2.322, Y 25.594, Z 33.150} C_DIS
   LIN {X -2.434, Y 26.676, Z 33.150} C_DIS
   LIN {X -2.849, Y 29.279, Z 33.150} C_DIS
   LIN {X -3.030, Y 30.388, Z 33.150} C_DIS
   LIN {X -3.329, Y 31.824, Z 33.150} C_DIS
   LIN {X -3.618, Y 33.224, Z 33.150} C_DIS
   LIN {X -3.896, Y 34.359, Z 33.150} C_DIS
   LIN {X -4.184, Y 35.527, Z 33.150} C_DIS
   LIN {X -4.392, Y 36.283, Z 33.150} C_DIS
   LIN {X -4.608, Y 37.070, Z 33.150} C_DIS
   LIN {X -4.734, Y 37.509, Z 33.150} C_DIS
   LIN {X -4.955, Y 38.272, Z 33.150} C_DIS
   LIN {X -5.113, Y 39.390, Z 33.150} C_DIS
   LIN {X -5.136, Y 39.553, Z 33.150} C_DIS
   LIN {X -5.109, Y 39.685, Z 33.150} C_DIS
   LIN {X -4.865, Y 40.898, Z 33.150} C_DIS
   LIN {X -4.012, Y 42.179, Z 33.150} C_DIS
   LIN {X -3.940, Y 42.287, Z 33.150} C_DIS
   LIN {X -3.340, Y 42.748, Z 33.150} C_DIS
   LIN {X -2.223, Y 43.147, Z 33.150} C_DIS
   LIN {X -1.263, Y 43.417, Z 33.150} C_DIS
   LIN {X -0.489, Y 43.263, Z 33.150} C_DIS
   LIN {X 0.450, Y 43.075, Z 33.150} C_DIS
   LIN {X 1.536, Y 42.273, Z 33.150} C_DIS
   LIN {X 1.851, Y 42.042, Z 33.150} C_DIS
   LIN {X 1.989, Y 41.809, Z 33.150} C_DIS
   LIN {X 2.600, Y 40.775, Z 33.150} C_DIS
   LIN {X 3.054, Y 39.509, Z 33.150} C_DIS
   LIN {X 3.101, Y 39.377, Z 33.150} C_DIS
   LIN {X 3.185, Y 39.130, Z 33.150} C_DIS
   LIN {X 3.723, Y 37.552, Z 33.150} C_DIS
   LIN {X 4.136, Y 36.265, Z 33.150} C_DIS
   LIN {X 4.456, Y 35.257, Z 33.150} C_DIS
   LIN {X 5.154, Y 32.845, Z 33.150} C_DIS
   LIN {X 5.372, Y 32.093, Z 33.150} C_DIS
   LIN {X 5.444, Y 31.852, Z 33.150} C_DIS
   LIN {X 5.515, Y 31.582, Z 33.150} C_DIS
   LIN {X 6.686, Y 26.697, Z 33.150} C_DIS
   LIN {X 7.461, Y 23.141, Z 33.150} C_DIS
   LIN {X 8.459, Y 16.543, Z 33.150} C_DIS
   LIN {X 8.648, Y 15.190, Z 33.150} C_DIS
   LIN {X 9.009, Y 11.714, Z 33.150} C_DIS
   LIN {X 9.297, Y 5.647, Z 33.150} C_DIS
   LIN {X 9.346, Y 3.606, Z 33.150} C_DIS
   LIN {X 9.153, Y -3.960, Z 33.150}
   LaserEnd_Ext()
   LIN {X -10.280, Y -19.895, Z 33.150}
   LaserStart_Ext()
   LIN {X -10.280, Y -24.630, Z 33.150}
   LaserEnd_Ext()
   LIN {X -9.280, Y -26.600, Z 33.150}
   LaserStart_Ext()
   LIN {X -9.280, Y -17.367, Z 33.150}
   LaserEnd_Ext()
   LIN {X -8.280, Y -15.415, Z 33.150}
   LaserStart_Ext()
   LIN {X -8.280, Y -20.444, Z 33.150}
   LaserEnd_Ext()
   LIN {X -8.280, Y -24.392, Z 33.150}
   LaserStart_Ext()
   LIN {X -8.280, Y -27.778, Z 33.150}
   LaserEnd_Ext()
   LIN {X -7.280, Y -28.618, Z 33.150}
   LaserStart_Ext()
   LIN {X -7.280, Y -26.057, Z 33.150}
   LaserEnd_Ext()
   LIN {X -7.280, Y -18.224, Z 33.150}
   LaserStart_Ext()
   LIN {X -7.280, Y -13.246, Z 33.150}
   LaserEnd_Ext()
   LIN {X -6.280, Y -10.961, Z 33.150}
   LaserStart_Ext()
   LIN {X -6.280, Y -17.433, Z 33.150}
   LaserEnd_Ext()
   LIN {X -6.280, Y -26.872, Z 33.150}
   LaserStart_Ext()
   LIN {X -6.280, Y -29.265, Z 33.150}
   LaserEnd_Ext()
   LIN {X -5.280, Y -29.609, Z 33.150}
   LaserStart_Ext()
   LIN {X -5.280, Y -27.573, Z 33.150}
   LaserEnd_Ext()
   LIN {X -5.280, Y -16.700, Z 33.150}
   LaserStart_Ext()
   LIN {X -5.280, Y -8.301, Z 33.150}
   LaserEnd_Ext()
   LIN {X -4.280, Y -5.389, Z 33.150}
   LaserStart_Ext()
   LIN {X -4.280, Y -16.442, Z 33.150}
   LaserEnd_Ext()
   LIN {X -4.280, Y -27.847, Z 33.150}
   LaserStart_Ext()
   LIN {X -4.280, Y -29.962, Z 33.150}
   LaserEnd_Ext()
   LIN {X -3.280, Y -30.027, Z 33.150}
   LaserStart_Ext()
   LIN {X -3.280, Y -28.042, Z 33.150}
   LaserEnd_Ext()
   LIN {X -3.280, Y -16.203, Z 33.150}
   LaserStart_Ext()
   LIN {X -3.280, Y -2.010, Z 33.150}
   LaserEnd_Ext()
   LIN {X -3.280, Y 36.011, Z 33.150}
   LaserStart_Ext()
   LIN {X -3.280, Y 41.474, Z 33.150}
   LaserEnd_Ext()
   LIN {X -2.280, Y 42.065, Z 33.150}
   LaserStart_Ext()
   LIN {X -2.280, Y 31.691, Z 33.150}
   LaserEnd_Ext()
   LIN {X -2.280, Y 2.521, Z 33.150}
   LaserStart_Ext()
   LIN {X -2.280, Y -16.220, Z 33.150}
   LaserEnd_Ext()
   LIN {X -2.280, Y -28.055, Z 33.150}
   LaserStart_Ext()
   LIN {X -2.280, Y -30.039, Z 33.150}
   LaserEnd_Ext()
   LIN {X -1.280, Y -29.898, Z 33.150}
   LaserStart_Ext()
   LIN {X -1.280, Y -27.821, Z 33.150}
   LaserEnd_Ext()
   LIN {X -1.280, Y -16.404, Z 33.150}
   LaserStart_Ext()
   LIN {X -1.280, Y 9.292, Z 33.150}
   LaserEnd_Ext()
   LIN {X -1.280, Y 25.236, Z 33.150}
   LaserStart_Ext()
   LIN {X -1.280, Y 42.373, Z 33.150}
   LaserEnd_Ext()
   LIN {X -0.280, Y 42.201, Z 33.150}
   LaserStart_Ext()
   LIN {X -0.280, Y -16.644, Z 33.150}
   LaserEnd_Ext()
   LIN {X -0.280, Y -27.583, Z 33.150}
   LaserStart_Ext()
   LIN {X -0.280, Y -29.527, Z 33.150}
   LaserEnd_Ext()
   LIN {X 0.720, Y -29.157, Z 33.150}
   LaserStart_Ext()
   LIN {X 0.720, Y -26.890, Z 33.150}
   LaserEnd_Ext()
   LIN {X 0.720, Y -17.346, Z 33.150}
   LaserStart_Ext()
   LIN {X 0.720, Y 41.632, Z 33.150}
   LaserEnd_Ext()
   LIN {X 1.720, Y 40.266, Z 33.150}
   LaserStart_Ext()
   LIN {X 1.720, Y -18.094, Z 33.150}
   LaserEnd_Ext()
   LIN {X 1.720, Y -26.106, Z 33.150}
   LaserStart_Ext()
   LIN {X 1.720, Y -28.651, Z 33.150}
   LaserEnd_Ext()
   LIN {X 2.720, Y -27.678, Z 33.150}
   LaserStart_Ext()
   LIN {X 2.720, Y -24.257, Z 33.150}
   LaserEnd_Ext()
   LIN {X 2.720, Y -19.952, Z 33.150}
   LaserStart_Ext()
   LIN {X 2.720, Y 37.395, Z 33.150}
   LaserEnd_Ext()
   LIN {X 3.720, Y 34.204, Z 33.150}
   LaserStart_Ext()
   LIN {X 3.720, Y -26.696, Z 33.150}
   LaserEnd_Ext()
   LIN {X 4.720, Y -24.692, Z 33.150}
   LaserStart_Ext()
   LIN {X 4.720, Y 30.609, Z 33.150}
   LaserEnd_Ext()
   LIN {X 5.720, Y 26.435, Z 33.150}
   LaserStart_Ext()
   LIN {X 5.720, Y -21.113, Z 33.150}
   LaserEnd_Ext()
   LIN {X 6.720, Y -15.999, Z 33.150}
   LaserStart_Ext()
   LIN {X 6.720, Y 21.353, Z 33.150}
   LaserEnd_Ext()
   LIN {X 7.720, Y 14.441, Z 33.150}
   LaserStart_Ext()
   LIN {X 7.720, Y -8.897, Z 33.150}
   LaserEnd_Ext()
   LIN {X -0.486, Y -26.573, Z 34.000}
   LaserStart_Ext()
   LIN {X -0.608, Y -26.603, Z 34.000} C_DIS
   LIN {X -2.630, Y -27.083, Z 34.000} C_DIS
   LIN {X -4.144, Y -26.795, Z 34.000} C_DIS
   LIN {X -4.640, Y -26.698, Z 34.000} C_DIS
   LIN {X -5.179, Y -26.319, Z 34.000} C_DIS
   LIN {X -6.332, Y -25.514, Z 34.000} C_DIS
   LIN {X -6.911, Y -24.559, Z 34.000} C_DIS
   LIN {X -7.409, Y -23.732, Z 34.000} C_DIS
   LIN {X -7.526, Y -22.722, Z 34.000} C_DIS
   LIN {X -7.652, Y -21.659, Z 34.000} C_DIS
   LIN {X -7.082, Y -20.291, Z 34.000} C_DIS
   LIN {X -6.477, Y -18.862, Z 34.000} C_DIS
   LIN {X -5.666, Y -18.239, Z 34.000} C_DIS
   LIN {X -4.816, Y -17.574, Z 34.000} C_DIS
   LIN {X -3.394, Y -17.229, Z 34.000} C_DIS
   LIN {X -2.779, Y -17.082, Z 34.000} C_DIS
   LIN {X -2.294, Y -17.172, Z 34.000} C_DIS
   LIN {X -0.707, Y -17.462, Z 34.000} C_DIS
   LIN {X 0.934, Y -18.620, Z 34.000} C_DIS
   LIN {X 1.029, Y -18.687, Z 34.000} C_DIS
   LIN {X 1.088, Y -18.801, Z 34.000} C_DIS
   LIN {X 2.213, Y -20.938, Z 34.000} C_DIS
   LIN {X 2.223, Y -22.781, Z 34.000} C_DIS
   LIN {X 2.223, Y -23.114, Z 34.000} C_DIS
   LIN {X 2.093, Y -23.374, Z 34.000} C_DIS
   LIN {X 1.141, Y -25.300, Z 34.000} C_DIS
   LIN {X -0.342, Y -26.460, Z 34.000} C_DIS
   LIN {X -0.486, Y -26.573, Z 34.000}
   LaserEnd_Ext()
   LIN {X 6.079, Y -24.217, Z 34.000}
   LaserStart_Ext()
   LIN {X 4.854, Y -26.998, Z 34.000} C_DIS
   LIN {X 3.043, Y -28.795, Z 34.000} C_DIS
   LIN {X 2.145, Y -29.669, Z 34.000} C_DIS
   LIN {X 0.082, Y -30.433, Z 34.000} C_DIS
   LIN {X -1.423, Y -30.999, Z 34.000} C_DIS
   LIN {X -3.051, Y -30.986, Z 34.000} C_DIS
   LIN {X -4.200, Y -30.972, Z 34.000} C_DIS
   LIN {X -4.547, Y -30.849, Z 34.000} C_DIS
   LIN {X -7.047, Y -29.988, Z 34.000} C_DIS
   LIN {X -9.315, Y -28.123, Z 34.000} C_DIS
   LIN {X -9.662, Y -27.812, Z 34.000} C_DIS
   LIN {X -9.914, Y -27.301, Z 34.000} C_DIS
   LIN {X -11.358, Y -24.542, Z 34.000} C_DIS
   LIN {X -11.567, Y -21.169, Z 34.000} C_DIS
   LIN {X -11.590, Y -20.839, Z 34.000} C_DIS
   LIN {X -11.441, Y -20.385, Z 34.000} C_DIS
   LIN {X -10.589, Y -17.830, Z 34.000} C_DIS
   LIN {X -9.577, Y -15.854, Z 34.000} C_DIS
   LIN {X -8.891, Y -14.498, Z 34.000} C_DIS
   LIN {X -8.285, Y -13.127, Z 34.000} C_DIS
   LIN {X -7.310, Y -10.945, Z 34.000} C_DIS
   LIN {X -5.950, Y -7.326, Z 34.000} C_DIS
   LIN {X -5.680, Y -6.611, Z 34.000} C_DIS
   LIN {X -5.546, Y -6.170, Z 34.000} C_DIS
   LIN {X -4.337, Y -2.223, Z 34.000} C_DIS
   LIN {X -3.013, Y 3.774, Z 34.000} C_DIS
   LIN {X -2.823, Y 4.647, Z 34.000} C_DIS
   LIN {X -2.702, Y 5.767, Z 34.000} C_DIS
   LIN {X -1.913, Y 12.617, Z 34.000} C_DIS
   LIN {X -1.893, Y 15.891, Z 34.000} C_DIS
   LIN {X -1.918, Y 21.103, Z 34.000} C_DIS
   LIN {X -2.155, Y 23.652, Z 34.000} C_DIS
   LIN {X -2.248, Y 24.548, Z 34.000} C_DIS
   LIN {X -2.453, Y 26.529, Z 34.000} C_DIS
   LIN {X -2.475, Y 26.741, Z 34.000} C_DIS
   LIN {X -2.500, Y 26.884, Z 34.000} C_DIS
   LIN {X -2.579, Y 27.368, Z 34.000} C_DIS
   LIN {X -3.077, Y 30.435, Z 34.000} C_DIS
   LIN {X -3.356, Y 31.771, Z 34.000} C_DIS
   LIN {X -3.673, Y 33.270, Z 34.000} C_DIS
   LIN {X -4.067, Y 34.854, Z 34.000} C_DIS
   LIN {X -4.243, Y 35.571, Z 34.000} C_DIS
   LIN {X -4.380, Y 36.066, Z 34.000} C_DIS
   LIN {X -4.671, Y 37.113, Z 34.000} C_DIS
   LIN {X -4.963, Y 38.115, Z 34.000} C_DIS
   LIN {X -5.021, Y 38.315, Z 34.000} C_DIS
   LIN {X -5.042, Y 38.466, Z 34.000} C_DIS
   LIN {X -5.205, Y 39.595, Z 34.000} C_DIS
   LIN {X -4.968, Y 40.782, Z 34.000} C_DIS
   LIN {X -4.926, Y 40.964, Z 34.000} C_DIS
   LIN {X -4.817, Y 41.123, Z 34.000} C_DIS
   LIN {X -4.014, Y 42.333, Z 34.000} C_DIS
   LIN {X -3.521, Y 42.712, Z 34.000} C_DIS
   LIN {X -2.153, Y 43.239, Z 34.000} C_DIS
   LIN {X -1.340, Y 43.468, Z 34.000} C_DIS
   LIN {X -0.440, Y 43.289, Z 34.000} C_DIS
   LIN {X 0.373, Y 43.130, Z 34.000} C_DIS
   LIN {X 0.713, Y 42.881, Z 34.000} C_DIS
   LIN {X 1.776, Y 42.100, Z 34.000} C_DIS
   LIN {X 2.456, Y 40.955, Z 34.000} C_DIS
   LIN {X 2.528, Y 40.835, Z 34.000} C_DIS
   LIN {X 2.569, Y 40.721, Z 34.000} C_DIS
   LIN {X 3.041, Y 39.413, Z 34.000} C_DIS
   LIN {X 3.525, Y 38.006, Z 34.000} C_DIS
   LIN {X 3.664, Y 37.600, Z 34.000} C_DIS
   LIN {X 3.906, Y 36.845, Z 34.000} C_DIS
   LIN {X 4.384, Y 35.365, Z 34.000} C_DIS
   LIN {X 4.945, Y 33.431, Z 34.000} C_DIS
   LIN {X 5.367, Y 32.011, Z 34.000} C_DIS
   LIN {X 5.784, Y 30.427, Z 34.000} C_DIS
   LIN {X 6.544, Y 27.257, Z 34.000} C_DIS
   LIN {X 7.469, Y 23.010, Z 34.000} C_DIS
   LIN {X 8.304, Y 17.493, Z 34.000} C_DIS
   LIN {X 8.715, Y 14.538, Z 34.000} C_DIS
   LIN {X 9.021, Y 11.597, Z 34.000} C_DIS
   LIN {X 9.340, Y 4.845, Z 34.000} C_DIS
   LIN {X 9.364, Y 3.877, Z 34.000} C_DIS
   LIN {X 9.253, Y -0.451, Z 34.000} C_DIS
   LIN {X 9.176, Y -4.090, Z 34.000} C_DIS
   LIN {X 9.052, Y -5.615, Z 34.000} C_DIS
   LIN {X 8.700, Y -9.636, Z 34.000} C_DIS
   LIN {X 8.200, Y -13.434, Z 34.000} C_DIS
   LIN {X 8.081, Y -14.296, Z 34.000} C_DIS
   LIN {X 7.921, Y -15.201, Z 34.000} C_DIS
   LIN {X 7.429, Y -18.073, Z 34.000} C_DIS
   LIN {X 7.104, Y -19.688, Z 34.000} C_DIS
   LIN {X 6.822, Y -21.039, Z 34.000} C_DIS
   LIN {X 6.118, Y -24.051, Z 34.000} C_DIS
   LIN {X 6.079, Y -24.217, Z 34.000}
   LaserEnd_Ext()
   LIN {X -5.799, Y -29.360, Z 34.000}
   LaserStart_Ext()
   LIN {X 0.100, Y -29.360, Z 34.000}
   LaserEnd_Ext()
   LIN {X 2.056, Y -28.360, Z 34.000}
   LaserStart_Ext()
   LIN {X -7.452, Y -28.360, Z 34.000}
   LaserEnd_Ext()
   LIN {X -8.668, Y -27.360, Z 34.000}
   LaserStart_Ext()
   LIN {X -5.437, Y -27.360, Z 34.000}
   LaserEnd_Ext()
   LIN {X 0.131, Y -27.360, Z 34.000}
   LaserStart_Ext()
   LIN {X 3.069, Y -27.360, Z 34.000}
   LaserEnd_Ext()
   LIN {X 4.042, Y -26.360, Z 34.000}
   LaserStart_Ext()
   LIN {X 1.409, Y -26.360, Z 34.000}
   LaserEnd_Ext()
   LIN {X -6.867, Y -26.360, Z 34.000}
   LaserStart_Ext()
   LIN {X -9.278, Y -26.360, Z 34.000}
   LaserEnd_Ext()
   LIN {X -9.801, Y -25.360, Z 34.000}
   LaserStart_Ext()
   LIN {X -7.595, Y -25.360, Z 34.000}
   LaserEnd_Ext()
   LIN {X 2.227, Y -25.360, Z 34.000}
   LaserStart_Ext()
   LIN {X 4.483, Y -25.360, Z 34.000}
   LaserEnd_Ext()
   LIN {X 4.924, Y -24.360, Z 34.000}
   LaserStart_Ext()
   LIN {X 2.721, Y -24.360, Z 34.000}
   LaserEnd_Ext()
   LIN {X -8.198, Y -24.360, Z 34.000}
   LaserStart_Ext()
   LIN {X -10.325, Y -24.360, Z 34.000}
   LaserEnd_Ext()
   LIN {X -10.430, Y -23.360, Z 34.000}
   LaserStart_Ext()
   LIN {X -8.458, Y -23.360, Z 34.000}
   LaserEnd_Ext()
   LIN {X 3.191, Y -23.360, Z 34.000}
   LaserStart_Ext()
   LIN {X 5.252, Y -23.360, Z 34.000}
   LaserEnd_Ext()
   LIN {X 5.486, Y -22.360, Z 34.000}
   LaserStart_Ext()
   LIN {X 3.221, Y -22.360, Z 34.000}
   LaserEnd_Ext()
   LIN {X -8.576, Y -22.360, Z 34.000}
   LaserStart_Ext()
   LIN {X -10.491, Y -22.360, Z 34.000}
   LaserEnd_Ext()
   LIN {X -10.553, Y -21.360, Z 34.000}
   LaserStart_Ext()
   LIN {X -8.606, Y -21.360, Z 34.000}
   LaserEnd_Ext()
   LIN {X 3.216, Y -21.360, Z 34.000}
   LaserStart_Ext()
   LIN {X 5.720, Y -21.360, Z 34.000}
   LaserEnd_Ext()
   LIN {X 5.942, Y -20.360, Z 34.000}
   LaserStart_Ext()
   LIN {X 3.039, Y -20.360, Z 34.000}
   LaserEnd_Ext()
   LIN {X -8.194, Y -20.360, Z 34.000}
   LaserStart_Ext()
   LIN {X -10.378, Y -20.360, Z 34.000}
   LaserEnd_Ext()
   LIN {X -10.045, Y -19.360, Z 34.000}
   LaserStart_Ext()
   LIN {X -7.774, Y -19.360, Z 34.000}
   LaserEnd_Ext()
   LIN {X 2.513, Y -19.360, Z 34.000}
   LaserStart_Ext()
   LIN {X 6.150, Y -19.360, Z 34.000}
   LaserEnd_Ext()
   LIN {X 6.351, Y -18.360, Z 34.000}
   LaserStart_Ext()
   LIN {X 1.986, Y -18.360, Z 34.000}
   LaserEnd_Ext()
   LIN {X -7.341, Y -18.360, Z 34.000}
   LaserStart_Ext()
   LIN {X -9.712, Y -18.360, Z 34.000}
   LaserEnd_Ext()
   LIN {X -9.225, Y -17.360, Z 34.000}
   LaserStart_Ext()
   LIN {X -6.165, Y -17.360, Z 34.000}
   LaserEnd_Ext()
   LIN {X 0.883, Y -17.360, Z 34.000}
   LaserStart_Ext()
   LIN {X 6.537, Y -17.360, Z 34.000}
   LaserEnd_Ext()
   LIN {X 6.708, Y -16.360, Z 34.000}
   LaserStart_Ext()
   LIN {X -1.174, Y -16.360, Z 34.000}
   LaserEnd_Ext()
   LIN {X -4.054, Y -16.360, Z 34.000}
   LaserStart_Ext()
   LIN {X -8.713, Y -16.360, Z 34.000}
   LaserEnd_Ext()
   LIN {X -8.207, Y -15.360, Z 34.000}
   LaserStart_Ext()
   LIN {X 6.880, Y -15.360, Z 34.000}
   LaserEnd_Ext()
   LIN {X 7.054, Y -14.360, Z 34.000}
   LaserStart_Ext()
   LIN {X -7.737, Y -14.360, Z 34.000}
   LaserEnd_Ext()
   LIN {X -7.294, Y -13.360, Z 34.000}
   LaserStart_Ext()
   LIN {X 7.200, Y -13.360, Z 34.000}
   LaserEnd_Ext()
   LIN {X 7.332, Y -12.360, Z 34.000}
   LaserStart_Ext()
   LIN {X -6.847, Y -12.360, Z 34.000}
   LaserEnd_Ext()
   LIN {X -6.401, Y -11.360, Z 34.000}
   LaserStart_Ext()
   LIN {X 7.464, Y -11.360, Z 34.000}
   LaserEnd_Ext()
   LIN {X 7.596, Y -10.360, Z 34.000}
   LaserStart_Ext()
   LIN {X -6.022, Y -10.360, Z 34.000}
   LaserEnd_Ext()
   LIN {X -5.646, Y -9.360, Z 34.000}
   LaserStart_Ext()
   LIN {X 7.720, Y -9.360, Z 34.000}
   LaserEnd_Ext()
   LIN {X 7.808, Y -8.360, Z 34.000}
   LaserStart_Ext()
   LIN {X -5.270, Y -8.360, Z 34.000}
   LaserEnd_Ext()
   LIN {X -4.894, Y -7.360, Z 34.000}
   LaserStart_Ext()
   LIN {X 7.895, Y -7.360, Z 34.000}
   LaserEnd_Ext()
   LIN {X 7.982, Y -6.360, Z 34.000}
   LaserStart_Ext()
   LIN {X -4.558, Y -6.360, Z 34.000}
   LaserEnd_Ext()
   LIN {X -4.252, Y -5.360, Z 34.000}
   LaserStart_Ext()
   LIN {X 8.069, Y -5.360, Z 34.000}
   LaserEnd_Ext()
   LIN {X 8.150, Y -4.360, Z 34.000}
   LaserStart_Ext()
   LIN {X -3.945, Y -4.360, Z 34.000}
   LaserEnd_Ext()
   LIN {X -3.639, Y -3.360, Z 34.000}
   LaserStart_Ext()
   LIN {X 8.191, Y -3.360, Z 34.000}
   LaserEnd_Ext()
   LIN {X 8.212, Y -2.360, Z 34.000}
   LaserStart_Ext()
   LIN {X -3.343, Y -2.360, Z 34.000}
   LaserEnd_Ext()
   LIN {X -3.122, Y -1.360, Z 34.000}
   LaserStart_Ext()
   LIN {X 8.234, Y -1.360, Z 34.000}
   LaserEnd_Ext()
   LIN {X 8.255, Y -0.360, Z 34.000}
   LaserStart_Ext()
   LIN {X -2.901, Y -0.360, Z 34.000}
   LaserEnd_Ext()
   LIN {X -2.681, Y 0.640, Z 34.000}
   LaserStart_Ext()
   LIN {X 8.281, Y 0.640, Z 34.000}
   LaserEnd_Ext()
   LIN {X 8.306, Y 1.640, Z 34.000}
   LaserStart_Ext()
   LIN {X -2.460, Y 1.640, Z 34.000}
   LaserEnd_Ext()
   LIN {X -2.239, Y 2.640, Z 34.000}
   LaserStart_Ext()
   LIN {X 8.332, Y 2.640, Z 34.000}
   LaserEnd_Ext()
   LIN {X 8.357, Y 3.640, Z 34.000}
   LaserStart_Ext()
   LIN {X -2.019, Y 3.640, Z 34.000}
   LaserEnd_Ext()
   LIN {X -1.818, Y 4.640, Z 34.000}
   LaserStart_Ext()
   LIN {X 8.345, Y 4.640, Z 34.000}
   LaserEnd_Ext()
   LIN {X 8.302, Y 5.640, Z 34.000}
   LaserStart_Ext()
   LIN {X -1.710, Y 5.640, Z 34.000}
   LaserEnd_Ext()
   LIN {X -1.594, Y 6.640, Z 34.000}
   LaserStart_Ext()
   LIN {X 8.254, Y 6.640, Z 34.000}
   LaserEnd_Ext()
   LIN {X 8.207, Y 7.640, Z 34.000}
   LaserStart_Ext()
   LIN {X -1.479, Y 7.640, Z 34.000}
   LaserEnd_Ext()
   LIN {X -1.364, Y 8.640, Z 34.000}
   LaserStart_Ext()
   LIN {X 8.160, Y 8.640, Z 34.000}
   LaserEnd_Ext()
   LIN {X 8.112, Y 9.640, Z 34.000}
   LaserStart_Ext()
   LIN {X -1.249, Y 9.640, Z 34.000}
   LaserEnd_Ext()
   LIN {X -1.134, Y 10.640, Z 34.000}
   LaserStart_Ext()
   LIN {X 8.065, Y 10.640, Z 34.000}
   LaserEnd_Ext()
   LIN {X 8.011, Y 11.640, Z 34.000}
   LaserStart_Ext()
   LIN {X -1.019, Y 11.640, Z 34.000}
   LaserEnd_Ext()
   LIN {X -0.913, Y 12.640, Z 34.000}
   LaserStart_Ext()
   LIN {X 7.907, Y 12.640, Z 34.000}
   LaserEnd_Ext()
   LIN {X 7.803, Y 13.640, Z 34.000}
   LaserStart_Ext()
   LIN {X -0.907, Y 13.640, Z 34.000}
   LaserEnd_Ext()
   LIN {X -0.900, Y 14.640, Z 34.000}
   LaserStart_Ext()
   LIN {X 7.691, Y 14.640, Z 34.000}
   LaserEnd_Ext()
   LIN {X 7.552, Y 15.640, Z 34.000}
   LaserStart_Ext()
   LIN {X -0.894, Y 15.640, Z 34.000}
   LaserEnd_Ext()
   LIN {X -0.897, Y 16.640, Z 34.000}
   LaserStart_Ext()
   LIN {X 7.413, Y 16.640, Z 34.000}
   LaserEnd_Ext()
   LIN {X 7.270, Y 17.640, Z 34.000}
   LaserStart_Ext()
   LIN {X -0.901, Y 17.640, Z 34.000}
   LaserEnd_Ext()
   LIN {X -0.906, Y 18.640, Z 34.000}
   LaserStart_Ext()
   LIN {X 7.119, Y 18.640, Z 34.000}
   LaserEnd_Ext()
   LIN {X 6.967, Y 19.640, Z 34.000}
   LaserStart_Ext()
   LIN {X -0.911, Y 19.640, Z 34.000}
   LaserEnd_Ext()
   LIN {X -0.916, Y 20.640, Z 34.000}
   LaserStart_Ext()
   LIN {X 6.816, Y 20.640, Z 34.000}
   LaserEnd_Ext()
   LIN {X 6.665, Y 21.640, Z 34.000}
   LaserStart_Ext()
   LIN {X -0.964, Y 21.640, Z 34.000}
   LaserEnd_Ext()
   LIN {X -1.057, Y 22.640, Z 34.000}
   LaserStart_Ext()
   LIN {X 6.513, Y 22.640, Z 34.000}
   LaserEnd_Ext()
   LIN {X 6.308, Y 23.640, Z 34.000}
   LaserStart_Ext()
   LIN {X -1.150, Y 23.640, Z 34.000}
   LaserEnd_Ext()
   LIN {X -1.252, Y 24.640, Z 34.000}
   LaserStart_Ext()
   LIN {X 6.090, Y 24.640, Z 34.000}
   LaserEnd_Ext()
   LIN {X 5.873, Y 25.640, Z 34.000}
   LaserStart_Ext()
   LIN {X -1.356, Y 25.640, Z 34.000}
   LaserEnd_Ext()
   LIN {X -1.459, Y 26.640, Z 34.000}
   LaserStart_Ext()
   LIN {X 5.655, Y 26.640, Z 34.000}
   LaserEnd_Ext()
   LIN {X 5.424, Y 27.640, Z 34.000}
   LaserStart_Ext()
   LIN {X -1.610, Y 27.640, Z 34.000}
   LaserEnd_Ext()
   LIN {X -1.772, Y 28.640, Z 34.000}
   LaserStart_Ext()
   LIN {X 5.184, Y 28.640, Z 34.000}
   LaserEnd_Ext()
   LIN {X 4.944, Y 29.640, Z 34.000}
   LaserStart_Ext()
   LIN {X -1.935, Y 29.640, Z 34.000}
   LaserEnd_Ext()
   LIN {X -2.099, Y 30.640, Z 34.000}
   LaserStart_Ext()
   LIN {X 4.694, Y 30.640, Z 34.000}
   LaserEnd_Ext()
   LIN {X 4.431, Y 31.640, Z 34.000}
   LaserStart_Ext()
   LIN {X -2.307, Y 31.640, Z 34.000}
   LaserEnd_Ext()
   LIN {X -2.517, Y 32.640, Z 34.000}
   LaserStart_Ext()
   LIN {X 4.137, Y 32.640, Z 34.000}
   LaserEnd_Ext()
   LIN {X 3.843, Y 33.640, Z 34.000}
   LaserStart_Ext()
   LIN {X -2.734, Y 33.640, Z 34.000}
   LaserEnd_Ext()
   LIN {X -2.983, Y 34.640, Z 34.000}
   LaserStart_Ext()
   LIN {X 3.553, Y 34.640, Z 34.000}
   LaserEnd_Ext()
   LIN {X 3.244, Y 35.640, Z 34.000}
   LaserStart_Ext()
   LIN {X -3.230, Y 35.640, Z 34.000}
   LaserEnd_Ext()
   LIN {X -3.501, Y 36.640, Z 34.000}
   LaserStart_Ext()
   LIN {X 2.922, Y 36.640, Z 34.000}
   LaserEnd_Ext()
   LIN {X 2.594, Y 37.640, Z 34.000}
   LaserStart_Ext()
   LIN {X -3.783, Y 37.640, Z 34.000}
   LaserEnd_Ext()
   LIN {X -4.057, Y 38.640, Z 34.000}
   LaserStart_Ext()
   LIN {X 2.250, Y 38.640, Z 34.000}
   LaserEnd_Ext()
   LIN {X 1.896, Y 39.640, Z 34.000}
   LaserStart_Ext()
   LIN {X -4.176, Y 39.640, Z 34.000}
   LaserEnd_Ext()
   LIN {X -3.937, Y 40.640, Z 34.000}
   LaserStart_Ext()
   LIN {X 1.480, Y 40.640, Z 34.000}
   LaserEnd_Ext()
   LIN {X 0.713, Y 41.640, Z 34.000}
   LaserStart_Ext()
   LIN {X -3.273, Y 41.640, Z 34.000}
   LaserEnd_Ext()
   LIN {X -6.425, Y -18.843, Z 34.850}
   LaserStart_Ext()
   LIN {X -6.127, Y -18.603, Z 34.850} C_DIS
   LIN {X -4.769, Y -17.540, Z 34.850} C_DIS
   LIN {X -3.510, Y -17.234, Z 34.850} C_DIS
   LIN {X -2.710, Y -17.034, Z 34.850} C_DIS
   LIN {X -1.673, Y -17.221, Z 34.850} C_DIS
   LIN {X -0.641, Y -17.410, Z 34.850} C_DIS
   LIN {X 0.061, Y -17.905, Z 34.850} C_DIS
   LIN {X 1.097, Y -18.630, Z 34.850} C_DIS
   LIN {X 1.864, Y -20.076, Z 34.850} C_DIS
   LIN {X 2.287, Y -20.878, Z 34.850} C_DIS
   LIN {X 2.291, Y -21.757, Z 34.850} C_DIS
   LIN {X 2.301, Y -23.054, Z 34.850} C_DIS
   LIN {X 1.231, Y -25.234, Z 34.850} C_DIS
   LIN {X -0.401, Y -26.521, Z 34.850} C_DIS
   LIN {X -1.790, Y -26.856, Z 34.850} C_DIS
   LIN {X -2.542, Y -27.035, Z 34.850} C_DIS
   LIN {X -3.530, Y -26.847, Z 34.850} C_DIS
   LIN {X -4.553, Y -26.655, Z 34.850} C_DIS
   LIN {X -5.192, Y -26.212, Z 34.850} C_DIS
   LIN {X -6.248, Y -25.475, Z 34.850} C_DIS
   LIN {X -7.090, Y -24.086, Z 34.850} C_DIS
   LIN {X -7.329, Y -23.695, Z 34.850} C_DIS
   LIN {X -7.382, Y -23.263, Z 34.850} C_DIS
   LIN {X -7.577, Y -21.623, Z 34.850} C_DIS
   LIN {X -6.608, Y -19.298, Z 34.850} C_DIS
   LIN {X -6.425, Y -18.843, Z 34.850}
   LaserEnd_Ext()
   LIN {X -10.866, Y -18.830, Z 34.850}
   LaserStart_Ext()
   LIN {X -10.523, Y -17.801, Z 34.850} C_DIS
   LIN {X -10.116, Y -17.005, Z 34.850} C_DIS
   LIN {X -8.861, Y -14.525, Z 34.850} C_DIS
   LIN {X -7.753, Y -12.017, Z 34.850} C_DIS
   LIN {X -7.302, Y -11.008, Z 34.850} C_DIS
   LIN {X -6.673, Y -9.335, Z 34.850} C_DIS
   LIN {X -5.718, Y -6.801, Z 34.850} C_DIS
   LIN {X -5.240, Y -5.238, Z 34.850} C_DIS
   LIN {X -4.335, Y -2.281, Z 34.850} C_DIS
   LIN {X -3.343, Y 2.212, Z 34.850} C_DIS
   LIN {X -2.827, Y 4.591, Z 34.850} C_DIS
   LIN {X -2.495, Y 7.642, Z 34.850} C_DIS
   LIN {X -1.922, Y 12.613, Z 34.850} C_DIS
   LIN {X -1.908, Y 14.989, Z 34.850} C_DIS
   LIN {X -1.938, Y 21.031, Z 34.850} C_DIS
   LIN {X -2.108, Y 22.860, Z 34.850} C_DIS
   LIN {X -2.174, Y 23.502, Z 34.850} C_DIS
   LIN {X -2.321, Y 24.923, Z 34.850} C_DIS
   LIN {X -2.534, Y 26.926, Z 34.850} C_DIS
   LIN {X -2.766, Y 28.274, Z 34.850} C_DIS
   LIN {X -3.125, Y 30.482, Z 34.850} C_DIS
   LIN {X -3.479, Y 32.142, Z 34.850} C_DIS
   LIN {X -3.727, Y 33.315, Z 34.850} C_DIS
   LIN {X -3.899, Y 34.009, Z 34.850} C_DIS
   LIN {X -4.303, Y 35.615, Z 34.850} C_DIS
   LIN {X -4.702, Y 37.041, Z 34.850} C_DIS
   LIN {X -4.734, Y 37.156, Z 34.850} C_DIS
   LIN {X -5.087, Y 38.357, Z 34.850} C_DIS
   LIN {X -5.241, Y 39.414, Z 34.850} C_DIS
   LIN {X -5.273, Y 39.645, Z 34.850} C_DIS
   LIN {X -5.185, Y 39.993, Z 34.850} C_DIS
   LIN {X -4.907, Y 41.211, Z 34.850} C_DIS
   LIN {X -4.307, Y 42.078, Z 34.850} C_DIS
   LIN {X -4.045, Y 42.417, Z 34.850} C_DIS
   LIN {X -3.668, Y 42.560, Z 34.850} C_DIS
   LIN {X -1.418, Y 43.518, Z 34.850} C_DIS
   LIN {X -0.519, Y 43.344, Z 34.850} C_DIS
   LIN {X 0.296, Y 43.184, Z 34.850} C_DIS
   LIN {X 1.539, Y 42.277, Z 34.850} C_DIS
   LIN {X 1.702, Y 42.158, Z 34.850} C_DIS
   LIN {X 1.757, Y 42.066, Z 34.850} C_DIS
   LIN {X 2.457, Y 40.894, Z 34.850} C_DIS
   LIN {X 2.926, Y 39.603, Z 34.850} C_DIS
   LIN {X 2.983, Y 39.446, Z 34.850} C_DIS
   LIN {X 3.079, Y 39.167, Z 34.850} C_DIS
   LIN {X 3.594, Y 37.680, Z 34.850} C_DIS
   LIN {X 4.039, Y 36.315, Z 34.850} C_DIS
   LIN {X 4.329, Y 35.415, Z 34.850} C_DIS
   LIN {X 4.517, Y 34.769, Z 34.850} C_DIS
   LIN {X 5.290, Y 32.170, Z 34.850} C_DIS
   LIN {X 6.052, Y 29.273, Z 34.850} C_DIS
   LIN {X 6.401, Y 27.817, Z 34.850} C_DIS
   LIN {X 7.477, Y 22.879, Z 34.850} C_DIS
   LIN {X 8.148, Y 18.443, Z 34.850} C_DIS
   LIN {X 8.782, Y 13.886, Z 34.850} C_DIS
   LIN {X 9.032, Y 11.481, Z 34.850} C_DIS
   LIN {X 9.373, Y 4.264, Z 34.850} C_DIS
   LIN {X 9.381, Y 4.129, Z 34.850} C_DIS
   LIN {X 9.377, Y 3.861, Z 34.850} C_DIS
   LIN {X 9.209, Y -4.033, Z 34.850} C_DIS
   LIN {X 8.914, Y -7.651, Z 34.850} C_DIS
   LIN {X 8.747, Y -9.562, Z 34.850} C_DIS
   LIN {X 8.352, Y -12.561, Z 34.850} C_DIS
   LIN {X 8.137, Y -14.234, Z 34.850} C_DIS
   LIN {X 8.008, Y -15.014, Z 34.850} C_DIS
   LIN {X 7.492, Y -18.024, Z 34.850} C_DIS
   LIN {X 6.959, Y -20.667, Z 34.850} C_DIS
   LIN {X 6.896, Y -20.969, Z 34.850} C_DIS
   LIN {X 6.738, Y -21.643, Z 34.850} C_DIS
   LIN {X 6.161, Y -24.148, Z 34.850} C_DIS
   LIN {X 5.624, Y -25.390, Z 34.850} C_DIS
   LIN {X 4.950, Y -26.920, Z 34.850} C_DIS
   LIN {X 2.505, Y -29.347, Z 34.850} C_DIS
   LIN {X 2.249, Y -29.604, Z 34.850} C_DIS
   LIN {X 2.059, Y -29.677, Z 34.850} C_DIS
   LIN {X -1.319, Y -30.947, Z 34.850} C_DIS
   LIN {X -3.579, Y -30.928, Z 34.850} C_DIS
   LIN {X -4.080, Y -30.931, Z 34.850} C_DIS
   LIN {X -5.129, Y -30.578, Z 34.850} C_DIS
   LIN {X -6.952, Y -29.951, Z 34.850} C_DIS
   LIN {X -8.589, Y -28.605, Z 34.850} C_DIS
   LIN {X -9.533, Y -27.834, Z 34.850} C_DIS
   LIN {X -9.916, Y -27.112, Z 34.850} C_DIS
   LIN {X -11.276, Y -24.515, Z 34.850} C_DIS
   LIN {X -11.416, Y -22.254, Z 34.850} C_DIS
   LIN {X -11.516, Y -20.812, Z 34.850} C_DIS
   LIN {X -10.866, Y -18.830, Z 34.850}
   LaserEnd_Ext()
   LIN {X 7.602, Y -10.594, Z 34.850}
   LaserStart_Ext()
   LIN {X 7.602, Y 15.108, Z 34.850}
   LaserEnd_Ext()
   LIN {X 6.602, Y 21.975, Z 34.850}
   LaserStart_Ext()
   LIN {X 6.602, Y -17.298, Z 34.850}
   LaserEnd_Ext()
   LIN {X 5.602, Y -22.121, Z 34.850}
   LaserStart_Ext()
   LIN {X 5.602, Y 26.787, Z 34.850}
   LaserEnd_Ext()
   LIN {X 4.602, Y 30.855, Z 34.850}
   LaserStart_Ext()
   LIN {X 4.602, Y -25.230, Z 34.850}
   LaserEnd_Ext()
   LIN {X 3.602, Y -26.849, Z 34.850}
   LaserStart_Ext()
   LIN {X 3.602, Y 34.337, Z 34.850}
   LaserEnd_Ext()
   LIN {X 2.602, Y 37.488, Z 34.850}
   LaserStart_Ext()
   LIN {X 2.602, Y -19.333, Z 34.850}
   LaserEnd_Ext()
   LIN {X 2.602, Y -24.711, Z 34.850}
   LaserStart_Ext()
   LIN {X 2.602, Y -27.842, Z 34.850}
   LaserEnd_Ext()
   LIN {X 1.602, Y -28.780, Z 34.850}
   LaserStart_Ext()
   LIN {X 1.602, Y -26.217, Z 34.850}
   LaserEnd_Ext()
   LIN {X 1.602, Y -17.763, Z 34.850}
   LaserStart_Ext()
   LIN {X 1.602, Y 40.318, Z 34.850}
   LaserEnd_Ext()
   LIN {X 0.602, Y 41.722, Z 34.850}
   LaserStart_Ext()
   LIN {X 0.602, Y -17.063, Z 34.850}
   LaserEnd_Ext()
   LIN {X 0.602, Y -27.004, Z 34.850}
   LaserStart_Ext()
   LIN {X 0.602, Y -29.156, Z 34.850}
   LaserEnd_Ext()
   LIN {X -0.398, Y -29.532, Z 34.850}
   LaserStart_Ext()
   LIN {X -0.398, Y -27.549, Z 34.850}
   LaserEnd_Ext()
   LIN {X -0.398, Y -16.441, Z 34.850}
   LaserStart_Ext()
   LIN {X -0.398, Y 42.302, Z 34.850}
   LaserEnd_Ext()
   LIN {X -1.398, Y 42.440, Z 34.850}
   LaserStart_Ext()
   LIN {X -1.398, Y 25.701, Z 34.850}
   LaserEnd_Ext()
   LIN {X -1.398, Y 8.425, Z 34.850}
   LaserStart_Ext()
   LIN {X -1.398, Y -16.255, Z 34.850}
   LaserEnd_Ext()
   LIN {X -1.398, Y -27.791, Z 34.850}
   LaserStart_Ext()
   LIN {X -1.398, Y -29.908, Z 34.850}
   LaserEnd_Ext()
   LIN {X -2.398, Y -29.938, Z 34.850}
   LaserStart_Ext()
   LIN {X -2.398, Y -28.024, Z 34.850}
   LaserEnd_Ext()
   LIN {X -2.398, Y -16.074, Z 34.850}
   LaserStart_Ext()
   LIN {X -2.398, Y 1.854, Z 34.850}
   LaserEnd_Ext()
   LIN {X -2.398, Y 31.869, Z 34.850}
   LaserStart_Ext()
   LIN {X -2.398, Y 42.014, Z 34.850}
   LaserEnd_Ext()
   LIN {X -3.398, Y 41.592, Z 34.850}
   LaserStart_Ext()
   LIN {X -3.398, Y 36.093, Z 34.850}
   LaserEnd_Ext()
   LIN {X -3.398, Y -2.638, Z 34.850}
   LaserStart_Ext()
   LIN {X -3.398, Y -16.176, Z 34.850}
   LaserEnd_Ext()
   LIN {X -3.398, Y -27.890, Z 34.850}
   LaserStart_Ext()
   LIN {X -3.398, Y -29.930, Z 34.850}
   LaserEnd_Ext()
   LIN {X -4.398, Y -29.769, Z 34.850}
   LaserStart_Ext()
   LIN {X -4.398, Y -27.701, Z 34.850}
   LaserEnd_Ext()
   LIN {X -4.398, Y -16.421, Z 34.850}
   LaserStart_Ext()
   LIN {X -4.398, Y -5.903, Z 34.850}
   LaserEnd_Ext()
   LIN {X -5.398, Y -8.787, Z 34.850}
   LaserStart_Ext()
   LIN {X -5.398, Y -16.762, Z 34.850}
   LaserEnd_Ext()
   LIN {X -5.398, Y -27.286, Z 34.850}
   LaserStart_Ext()
   LIN {X -5.398, Y -29.428, Z 34.850}
   LaserEnd_Ext()
   LIN {X -6.398, Y -29.084, Z 34.850}
   LaserStart_Ext()
   LIN {X -6.398, Y -26.590, Z 34.850}
   LaserEnd_Ext()
   LIN {X -6.398, Y -17.545, Z 34.850}
   LaserStart_Ext()
   LIN {X -6.398, Y -11.436, Z 34.850}
   LaserEnd_Ext()
   LIN {X -7.398, Y -13.688, Z 34.850}
   LaserStart_Ext()
   LIN {X -7.398, Y -18.582, Z 34.850}
   LaserEnd_Ext()
   LIN {X -7.398, Y -25.507, Z 34.850}
   LaserStart_Ext()
   LIN {X -7.398, Y -28.289, Z 34.850}
   LaserEnd_Ext()
   LIN {X -8.398, Y -27.469, Z 34.850}
   LaserStart_Ext()
   LIN {X -8.398, Y -23.187, Z 34.850}
   LaserEnd_Ext()
   LIN {X -8.398, Y -20.993, Z 34.850}
   LaserStart_Ext()
   LIN {X -8.398, Y -15.825, Z 34.850}
   LaserEnd_Ext()
   LIN {X -9.398, Y -17.798, Z 34.850}
   LaserStart_Ext()
   LIN {X -9.398, Y -25.946, Z 34.850}
   LaserEnd_Ext()
   LIN {X -10.398, Y -22.512, Z 34.850}
   LaserStart_Ext()
   LIN {X -10.398, Y -20.611, Z 34.850}
   LaserEnd_Ext()
   LIN {X -1.674, Y -26.797, Z 35.700}
   LaserStart_Ext()
   LIN {X -2.454, Y -26.987, Z 35.700} C_DIS
   LIN {X -2.956, Y -26.895, Z 35.700} C_DIS
   LIN {X -4.466, Y -26.611, Z 35.700} C_DIS
   LIN {X -6.148, Y -25.446, Z 35.700} C_DIS
   LIN {X -7.249, Y -23.658, Z 35.700} C_DIS
   LIN {X -7.486, Y -21.722, Z 35.700} C_DIS
   LIN {X -7.502, Y -21.586, Z 35.700} C_DIS
   LIN {X -7.422, Y -21.394, Z 35.700} C_DIS
   LIN {X -6.399, Y -18.857, Z 35.700} C_DIS
   LIN {X -4.738, Y -17.518, Z 35.700} C_DIS
   LIN {X -2.646, Y -16.986, Z 35.700} C_DIS
   LIN {X -1.061, Y -17.272, Z 35.700} C_DIS
   LIN {X -0.576, Y -17.357, Z 35.700} C_DIS
   LIN {X -0.072, Y -17.707, Z 35.700} C_DIS
   LIN {X 1.165, Y -18.574, Z 35.700} C_DIS
   LIN {X 1.942, Y -20.038, Z 35.700} C_DIS
   LIN {X 2.360, Y -20.819, Z 35.700} C_DIS
   LIN {X 2.368, Y -21.495, Z 35.700} C_DIS
   LIN {X 2.380, Y -22.995, Z 35.700} C_DIS
   LIN {X 1.824, Y -24.126, Z 35.700} C_DIS
   LIN {X 1.311, Y -25.183, Z 35.700} C_DIS
   LIN {X 0.360, Y -25.937, Z 35.700} C_DIS
   LIN {X -0.316, Y -26.468, Z 35.700} C_DIS
   LIN {X -1.674, Y -26.797, Z 35.700}
   LaserEnd_Ext()
   LIN {X -0.669, Y 43.409, Z 35.700}
   LaserStart_Ext()
   LIN {X -1.495, Y 43.569, Z 35.700} C_DIS
   LIN {X -2.090, Y 43.315, Z 35.700} C_DIS
   LIN {X -3.955, Y 42.611, Z 35.700} C_DIS
   LIN {X -4.467, Y 41.948, Z 35.700} C_DIS
   LIN {X -4.915, Y 41.394, Z 35.700} C_DIS
   LIN {X -5.048, Y 40.892, Z 35.700} C_DIS
   LIN {X -5.340, Y 39.737, Z 35.700} C_DIS
   LIN {X -5.191, Y 38.676, Z 35.700} C_DIS
   LIN {X -5.153, Y 38.399, Z 35.700} C_DIS
   LIN {X -5.089, Y 38.187, Z 35.700} C_DIS
   LIN {X -4.796, Y 37.199, Z 35.700} C_DIS
   LIN {X -4.446, Y 35.960, Z 35.700} C_DIS
   LIN {X -4.362, Y 35.659, Z 35.700} C_DIS
   LIN {X -4.219, Y 35.088, Z 35.700} C_DIS
   LIN {X -3.780, Y 33.360, Z 35.700} C_DIS
   LIN {X -3.463, Y 31.894, Z 35.700} C_DIS
   LIN {X -3.172, Y 30.529, Z 35.700} C_DIS
   LIN {X -3.031, Y 29.664, Z 35.700} C_DIS
   LIN {X -2.593, Y 27.111, Z 35.700} C_DIS
   LIN {X -2.189, Y 23.317, Z 35.700} C_DIS
   LIN {X -2.100, Y 22.456, Z 35.700} C_DIS
   LIN {X -2.060, Y 22.067, Z 35.700} C_DIS
   LIN {X -1.957, Y 20.959, Z 35.700} C_DIS
   LIN {X -1.923, Y 14.087, Z 35.700} C_DIS
   LIN {X -1.932, Y 12.609, Z 35.700} C_DIS
   LIN {X -2.288, Y 9.517, Z 35.700} C_DIS
   LIN {X -2.830, Y 4.534, Z 35.700} C_DIS
   LIN {X -3.673, Y 0.650, Z 35.700} C_DIS
   LIN {X -4.333, Y -2.338, Z 35.700} C_DIS
   LIN {X -4.935, Y -4.305, Z 35.700} C_DIS
   LIN {X -5.757, Y -6.990, Z 35.700} C_DIS
   LIN {X -7.189, Y -10.793, Z 35.700} C_DIS
   LIN {X -7.286, Y -11.054, Z 35.700} C_DIS
   LIN {X -7.364, Y -11.233, Z 35.700} C_DIS
   LIN {X -8.831, Y -14.553, Z 35.700} C_DIS
   LIN {X -10.298, Y -17.453, Z 35.700} C_DIS
   LIN {X -10.457, Y -17.772, Z 35.700} C_DIS
   LIN {X -10.556, Y -18.081, Z 35.700} C_DIS
   LIN {X -11.443, Y -20.785, Z 35.700} C_DIS
   LIN {X -11.265, Y -23.339, Z 35.700} C_DIS
   LIN {X -11.194, Y -24.487, Z 35.700} C_DIS
   LIN {X -10.503, Y -25.807, Z 35.700} C_DIS
   LIN {X -9.443, Y -27.802, Z 35.700} C_DIS
   LIN {X -6.867, Y -29.905, Z 35.700} C_DIS
   LIN {X -3.947, Y -30.891, Z 35.700} C_DIS
   LIN {X -2.545, Y -30.884, Z 35.700} C_DIS
   LIN {X -1.214, Y -30.895, Z 35.700} C_DIS
   LIN {X 0.774, Y -30.147, Z 35.700} C_DIS
   LIN {X 2.349, Y -29.540, Z 35.700} C_DIS
   LIN {X 4.469, Y -27.415, Z 35.700} C_DIS
   LIN {X 5.045, Y -26.843, Z 35.700} C_DIS
   LIN {X 5.205, Y -26.482, Z 35.700} C_DIS
   LIN {X 6.242, Y -24.079, Z 35.700} C_DIS
   LIN {X 6.782, Y -21.739, Z 35.700} C_DIS
   LIN {X 6.970, Y -20.899, Z 35.700} C_DIS
   LIN {X 7.212, Y -19.674, Z 35.700} C_DIS
   LIN {X 7.555, Y -17.974, Z 35.700} C_DIS
   LIN {X 7.809, Y -16.488, Z 35.700} C_DIS
   LIN {X 8.195, Y -14.160, Z 35.700} C_DIS
   LIN {X 8.773, Y -9.655, Z 35.700} C_DIS
   LIN {X 8.793, Y -9.489, Z 35.700} C_DIS
   LIN {X 8.814, Y -9.221, Z 35.700} C_DIS
   LIN {X 9.241, Y -3.975, Z 35.700} C_DIS
   LIN {X 9.351, Y 1.158, Z 35.700} C_DIS
   LIN {X 9.395, Y 4.214, Z 35.700} C_DIS
   LIN {X 9.309, Y 5.755, Z 35.700} C_DIS
   LIN {X 9.043, Y 11.365, Z 35.700} C_DIS
   LIN {X 8.848, Y 13.235, Z 35.700} C_DIS
   LIN {X 7.992, Y 19.393, Z 35.700} C_DIS
   LIN {X 7.484, Y 22.747, Z 35.700} C_DIS
   LIN {X 6.337, Y 28.016, Z 35.700} C_DIS
   LIN {X 6.272, Y 28.308, Z 35.700} C_DIS
   LIN {X 6.128, Y 28.850, Z 35.700} C_DIS
   LIN {X 5.213, Y 32.329, Z 35.700} C_DIS
   LIN {X 4.583, Y 34.445, Z 35.700} C_DIS
   LIN {X 4.268, Y 35.486, Z 35.700} C_DIS
   LIN {X 3.777, Y 36.982, Z 35.700} C_DIS
   LIN {X 3.520, Y 37.770, Z 35.700} C_DIS
   LIN {X 3.379, Y 38.179, Z 35.700} C_DIS
   LIN {X 2.907, Y 39.527, Z 35.700} C_DIS
   LIN {X 2.401, Y 40.909, Z 35.700} C_DIS
   LIN {X 1.628, Y 42.215, Z 35.700} C_DIS
   LIN {X 0.670, Y 42.913, Z 35.700} C_DIS
   LIN {X 0.220, Y 43.239, Z 35.700} C_DIS
   LIN {X -0.669, Y 43.409, Z 35.700}
   LaserEnd_Ext()
   LIN {X -1.347, Y 42.522, Z 35.700}
   LaserStart_Ext()
   LIN {X -1.402, Y 42.522, Z 35.700}
   LaserEnd_Ext()
   LIN {X -3.533, Y 41.522, Z 35.700}
   LaserStart_Ext()
   LIN {X 0.878, Y 41.522, Z 35.700}
   LaserEnd_Ext()
   LIN {X 1.478, Y 40.522, Z 35.700}
   LaserStart_Ext()
   LIN {X -4.110, Y 40.522, Z 35.700}
   LaserEnd_Ext()
   LIN {X -4.300, Y 39.522, Z 35.700}
   LaserStart_Ext()
   LIN {X 1.844, Y 39.522, Z 35.700}
   LaserEnd_Ext()
   LIN {X 2.199, Y 38.522, Z 35.700}
   LaserStart_Ext()
   LIN {X -4.146, Y 38.522, Z 35.700}
   LaserEnd_Ext()
   LIN {X -3.849, Y 37.522, Z 35.700}
   LaserStart_Ext()
   LIN {X 2.548, Y 37.522, Z 35.700}
   LaserEnd_Ext()
   LIN {X 2.876, Y 36.522, Z 35.700}
   LaserStart_Ext()
   LIN {X -3.566, Y 36.522, Z 35.700}
   LaserEnd_Ext()
   LIN {X -3.296, Y 35.522, Z 35.700}
   LaserStart_Ext()
   LIN {X 3.204, Y 35.522, Z 35.700}
   LaserEnd_Ext()
   LIN {X 3.515, Y 34.522, Z 35.700}
   LaserStart_Ext()
   LIN {X -3.043, Y 34.522, Z 35.700}
   LaserEnd_Ext()
   LIN {X -2.792, Y 33.522, Z 35.700}
   LaserStart_Ext()
   LIN {X 3.815, Y 33.522, Z 35.700}
   LaserEnd_Ext()
   LIN {X 4.112, Y 32.522, Z 35.700}
   LaserStart_Ext()
   LIN {X -2.576, Y 32.522, Z 35.700}
   LaserEnd_Ext()
   LIN {X -2.361, Y 31.522, Z 35.700}
   LaserStart_Ext()
   LIN {X 4.391, Y 31.522, Z 35.700}
   LaserEnd_Ext()
   LIN {X 4.654, Y 30.522, Z 35.700}
   LaserStart_Ext()
   LIN {X -2.158, Y 30.522, Z 35.700}
   LaserEnd_Ext()
   LIN {X -1.992, Y 29.522, Z 35.700}
   LaserStart_Ext()
   LIN {X 4.917, Y 29.522, Z 35.700}
   LaserEnd_Ext()
   LIN {X 5.181, Y 28.522, Z 35.700}
   LaserStart_Ext()
   LIN {X -1.821, Y 28.522, Z 35.700}
   LaserEnd_Ext()
   LIN {X -1.649, Y 27.522, Z 35.700}
   LaserStart_Ext()
   LIN {X 5.421, Y 27.522, Z 35.700}
   LaserEnd_Ext()
   LIN {X 5.639, Y 26.522, Z 35.700}
   LaserStart_Ext()
   LIN {X -1.525, Y 26.522, Z 35.700}
   LaserEnd_Ext()
   LIN {X -1.418, Y 25.522, Z 35.700}
   LaserStart_Ext()
   LIN {X 5.857, Y 25.522, Z 35.700}
   LaserEnd_Ext()
   LIN {X 6.075, Y 24.522, Z 35.700}
   LaserStart_Ext()
   LIN {X -1.312, Y 24.522, Z 35.700}
   LaserEnd_Ext()
   LIN {X -1.205, Y 23.522, Z 35.700}
   LaserStart_Ext()
   LIN {X 6.292, Y 23.522, Z 35.700}
   LaserEnd_Ext()
   LIN {X 6.507, Y 22.522, Z 35.700}
   LaserStart_Ext()
   LIN {X -1.101, Y 22.522, Z 35.700}
   LaserEnd_Ext()
   LIN {X -1.005, Y 21.522, Z 35.700}
   LaserStart_Ext()
   LIN {X 6.659, Y 21.522, Z 35.700}
   LaserEnd_Ext()
   LIN {X 6.810, Y 20.522, Z 35.700}
   LaserStart_Ext()
   LIN {X -0.955, Y 20.522, Z 35.700}
   LaserEnd_Ext()
   LIN {X -0.950, Y 19.522, Z 35.700}
   LaserStart_Ext()
   LIN {X 6.961, Y 19.522, Z 35.700}
   LaserEnd_Ext()
   LIN {X 7.104, Y 18.522, Z 35.700}
   LaserStart_Ext()
   LIN {X -0.945, Y 18.522, Z 35.700}
   LaserEnd_Ext()
   LIN {X -0.940, Y 17.522, Z 35.700}
   LaserStart_Ext()
   LIN {X 7.243, Y 17.522, Z 35.700}
   LaserEnd_Ext()
   LIN {X 7.382, Y 16.522, Z 35.700}
   LaserStart_Ext()
   LIN {X -0.935, Y 16.522, Z 35.700}
   LaserEnd_Ext()
   LIN {X -0.930, Y 15.522, Z 35.700}
   LaserStart_Ext()
   LIN {X 7.521, Y 15.522, Z 35.700}
   LaserEnd_Ext()
   LIN {X 7.660, Y 14.522, Z 35.700}
   LaserStart_Ext()
   LIN {X -0.925, Y 14.522, Z 35.700}
   LaserEnd_Ext()
   LIN {X -0.926, Y 13.522, Z 35.700}
   LaserStart_Ext()
   LIN {X 7.799, Y 13.522, Z 35.700}
   LaserEnd_Ext()
   LIN {X 7.917, Y 12.522, Z 35.700}
   LaserStart_Ext()
   LIN {X -0.937, Y 12.522, Z 35.700}
   LaserEnd_Ext()
   LIN {X -1.051, Y 11.522, Z 35.700}
   LaserStart_Ext()
   LIN {X 8.021, Y 11.522, Z 35.700}
   LaserEnd_Ext()
   LIN {X 8.082, Y 10.522, Z 35.700}
   LaserStart_Ext()
   LIN {X -1.166, Y 10.522, Z 35.700}
   LaserEnd_Ext()
   LIN {X -1.281, Y 9.522, Z 35.700}
   LaserStart_Ext()
   LIN {X 8.129, Y 9.522, Z 35.700}
   LaserEnd_Ext()
   LIN {X 8.177, Y 8.522, Z 35.700}
   LaserStart_Ext()
   LIN {X -1.391, Y 8.522, Z 35.700}
   LaserEnd_Ext()
   LIN {X -1.499, Y 7.522, Z 35.700}
   LaserStart_Ext()
   LIN {X 8.224, Y 7.522, Z 35.700}
   LaserEnd_Ext()
   LIN {X 8.271, Y 6.522, Z 35.700}
   LaserStart_Ext()
   LIN {X -1.608, Y 6.522, Z 35.700}
   LaserEnd_Ext()
   LIN {X -1.717, Y 5.522, Z 35.700}
   LaserStart_Ext()
   LIN {X 8.320, Y 5.522, Z 35.700}
   LaserEnd_Ext()
   LIN {X 8.377, Y 4.522, Z 35.700}
   LaserStart_Ext()
   LIN {X -1.825, Y 4.522, Z 35.700}
   LaserEnd_Ext()
   LIN {X -2.027, Y 3.522, Z 35.700}
   LaserStart_Ext()
   LIN {X 8.385, Y 3.522, Z 35.700}
   LaserEnd_Ext()
   LIN {X 8.371, Y 2.522, Z 35.700}
   LaserStart_Ext()
   LIN {X -2.244, Y 2.522, Z 35.700}
   LaserEnd_Ext()
   LIN {X -2.461, Y 1.522, Z 35.700}
   LaserStart_Ext()
   LIN {X 8.356, Y 1.522, Z 35.700}
   LaserEnd_Ext()
   LIN {X 8.337, Y 0.522, Z 35.700}
   LaserStart_Ext()
   LIN {X -2.678, Y 0.522, Z 35.700}
   LaserEnd_Ext()
   LIN {X -2.898, Y -0.478, Z 35.700}
   LaserStart_Ext()
   LIN {X 8.316, Y -0.478, Z 35.700}
   LaserEnd_Ext()
   LIN {X 8.294, Y -1.478, Z 35.700}
   LaserStart_Ext()
   LIN {X -3.119, Y -1.478, Z 35.700}
   LaserEnd_Ext()
   LIN {X -3.340, Y -2.478, Z 35.700}
   LaserStart_Ext()
   LIN {X 8.273, Y -2.478, Z 35.700}
   LaserEnd_Ext()
   LIN {X 8.252, Y -3.478, Z 35.700}
   LaserStart_Ext()
   LIN {X -3.636, Y -3.478, Z 35.700}
   LaserEnd_Ext()
   LIN {X -3.942, Y -4.478, Z 35.700}
   LaserStart_Ext()
   LIN {X 8.197, Y -4.478, Z 35.700}
   LaserEnd_Ext()
   LIN {X 8.116, Y -5.478, Z 35.700}
   LaserStart_Ext()
   LIN {X -4.248, Y -5.478, Z 35.700}
   LaserEnd_Ext()
   LIN {X -4.554, Y -6.478, Z 35.700}
   LaserStart_Ext()
   LIN {X 8.034, Y -6.478, Z 35.700}
   LaserEnd_Ext()
   LIN {X 7.953, Y -7.478, Z 35.700}
   LaserStart_Ext()
   LIN {X -4.872, Y -7.478, Z 35.700}
   LaserEnd_Ext()
   LIN {X -5.248, Y -8.478, Z 35.700}
   LaserStart_Ext()
   LIN {X 7.871, Y -8.478, Z 35.700}
   LaserEnd_Ext()
   LIN {X 7.787, Y -9.478, Z 35.700}
   LaserStart_Ext()
   LIN {X -5.625, Y -9.478, Z 35.700}
   LaserEnd_Ext()
   LIN {X -6.002, Y -10.478, Z 35.700}
   LaserStart_Ext()
   LIN {X 7.659, Y -10.478, Z 35.700}
   LaserEnd_Ext()
   LIN {X 7.531, Y -11.478, Z 35.700}
   LaserStart_Ext()
   LIN {X -6.381, Y -11.478, Z 35.700}
   LaserEnd_Ext()
   LIN {X -6.821, Y -12.478, Z 35.700}
   LaserStart_Ext()
   LIN {X 7.402, Y -12.478, Z 35.700}
   LaserEnd_Ext()
   LIN {X 7.274, Y -13.478, Z 35.700}
   LaserStart_Ext()
   LIN {X -7.263, Y -13.478, Z 35.700}
   LaserEnd_Ext()
   LIN {X -7.705, Y -14.478, Z 35.700}
   LaserStart_Ext()
   LIN {X 7.129, Y -14.478, Z 35.700}
   LaserEnd_Ext()
   LIN {X 6.963, Y -15.478, Z 35.700}
   LaserStart_Ext()
   LIN {X -8.179, Y -15.478, Z 35.700}
   LaserEnd_Ext()
   LIN {X -8.685, Y -16.478, Z 35.700}
   LaserStart_Ext()
   LIN {X -4.735, Y -16.478, Z 35.700}
   LaserEnd_Ext()
   LIN {X -0.099, Y -16.478, Z 35.700}
   LaserStart_Ext()
   LIN {X 6.797, Y -16.478, Z 35.700}
   LaserEnd_Ext()
   LIN {X 6.625, Y -17.478, Z 35.700}
   LaserStart_Ext()
   LIN {X 1.344, Y -17.478, Z 35.700}
   LaserEnd_Ext()
   LIN {X -6.282, Y -17.478, Z 35.700}
   LaserStart_Ext()
   LIN {X -9.190, Y -17.478, Z 35.700}
   LaserEnd_Ext()
   LIN {X -9.634, Y -18.478, Z 35.700}
   LaserStart_Ext()
   LIN {X -7.325, Y -18.478, Z 35.700}
   LaserEnd_Ext()
   LIN {X 2.247, Y -18.478, Z 35.700}
   LaserStart_Ext()
   LIN {X 6.433, Y -18.478, Z 35.700}
   LaserEnd_Ext()
   LIN {X 6.231, Y -19.478, Z 35.700}
   LaserStart_Ext()
   LIN {X 2.777, Y -19.478, Z 35.700}
   LaserEnd_Ext()
   LIN {X -7.728, Y -19.478, Z 35.700}
   LaserStart_Ext()
   LIN {X -9.962, Y -19.478, Z 35.700}
   LaserEnd_Ext()
   LIN {X -10.290, Y -20.478, Z 35.700}
   LaserStart_Ext()
   LIN {X -8.131, Y -20.478, Z 35.700}
   LaserEnd_Ext()
   LIN {X 3.299, Y -20.478, Z 35.700}
   LaserStart_Ext()
   LIN {X 6.034, Y -20.478, Z 35.700}
   LaserEnd_Ext()
   LIN {X 5.815, Y -21.478, Z 35.700}
   LaserStart_Ext()
   LIN {X 3.368, Y -21.478, Z 35.700}
   LaserEnd_Ext()
   LIN {X -8.496, Y -21.478, Z 35.700}
   LaserStart_Ext()
   LIN {X -10.392, Y -21.478, Z 35.700}
   LaserEnd_Ext()
   LIN {X -10.323, Y -22.478, Z 35.700}
   LaserStart_Ext()
   LIN {X -8.401, Y -22.478, Z 35.700}
   LaserEnd_Ext()
   LIN {X 3.376, Y -22.478, Z 35.700}
   LaserStart_Ext()
   LIN {X 5.585, Y -22.478, Z 35.700}
   LaserEnd_Ext()
   LIN {X 5.355, Y -23.478, Z 35.700}
   LaserStart_Ext()
   LIN {X 3.257, Y -23.478, Z 35.700}
   LaserEnd_Ext()
   LIN {X -8.279, Y -23.478, Z 35.700}
   LaserStart_Ext()
   LIN {X -10.255, Y -23.478, Z 35.700}
   LaserEnd_Ext()
   LIN {X -10.070, Y -24.478, Z 35.700}
   LaserStart_Ext()
   LIN {X -7.920, Y -24.478, Z 35.700}
   LaserEnd_Ext()
   LIN {X 2.765, Y -24.478, Z 35.700}
   LaserStart_Ext()
   LIN {X 4.981, Y -24.478, Z 35.700}
   LaserEnd_Ext()
   LIN {X 4.549, Y -25.478, Z 35.700}
   LaserStart_Ext()
   LIN {X 2.279, Y -25.478, Z 35.700}
   LaserEnd_Ext()
   LIN {X -7.309, Y -25.478, Z 35.700}
   LaserStart_Ext()
   LIN {X -9.546, Y -25.478, Z 35.700}
   LaserEnd_Ext()
   LIN {X -9.014, Y -26.478, Z 35.700}
   LaserStart_Ext()
   LIN {X -6.414, Y -26.478, Z 35.700}
   LaserEnd_Ext()
   LIN {X 1.286, Y -26.478, Z 35.700}
   LaserStart_Ext()
   LIN {X 3.993, Y -26.478, Z 35.700}
   LaserEnd_Ext()
   LIN {X 2.993, Y -27.478, Z 35.700}
   LaserStart_Ext()
   LIN {X -0.238, Y -27.478, Z 35.700}
   LaserEnd_Ext()
   LIN {X -4.962, Y -27.478, Z 35.700}
   LaserStart_Ext()
   LIN {X -8.258, Y -27.478, Z 35.700}
   LaserEnd_Ext()
   LIN {X -7.034, Y -28.478, Z 35.700}
   LaserStart_Ext()
   LIN {X 1.996, Y -28.478, Z 35.700}
   LaserEnd_Ext()
   LIN {X -0.288, Y -29.478, Z 35.700}
   LaserStart_Ext()
   LIN {X -5.013, Y -29.478, Z 35.700}
   LaserEnd_Ext()
   LIN {X -6.080, Y -25.396, Z 36.550}
   LaserStart_Ext()
   LIN {X -6.778, Y -24.261, Z 36.550} C_DIS
   LIN {X -7.169, Y -23.621, Z 36.550} C_DIS
   LIN {X -7.265, Y -22.837, Z 36.550} C_DIS
   LIN {X -7.427, Y -21.550, Z 36.550} C_DIS
   LIN {X -6.700, Y -19.679, Z 36.550} C_DIS
   LIN {X -6.374, Y -18.872, Z 36.550} C_DIS
   LIN {X -5.905, Y -18.494, Z 36.550} C_DIS
   LIN {X -4.756, Y -17.518, Z 36.550} C_DIS
   LIN {X -2.938, Y -17.028, Z 36.550} C_DIS
   LIN {X -2.582, Y -16.939, Z 36.550} C_DIS
   LIN {X -2.313, Y -16.987, Z 36.550} C_DIS
   LIN {X -0.511, Y -17.304, Z 36.550} C_DIS
   LIN {X 1.129, Y -18.445, Z 36.550} C_DIS
   LIN {X 1.233, Y -18.517, Z 36.550} C_DIS
   LIN {X 1.311, Y -18.661, Z 36.550} C_DIS
   LIN {X 2.434, Y -20.759, Z 36.550} C_DIS
   LIN {X 2.458, Y -22.832, Z 36.550} C_DIS
   LIN {X 2.458, Y -22.935, Z 36.550} C_DIS
   LIN {X 1.393, Y -25.128, Z 36.550} C_DIS
   LIN {X 0.212, Y -26.063, Z 36.550} C_DIS
   LIN {X -0.232, Y -26.416, Z 36.550} C_DIS
   LIN {X -0.593, Y -26.506, Z 36.550} C_DIS
   LIN {X -2.366, Y -26.938, Z 36.550} C_DIS
   LIN {X -4.101, Y -26.620, Z 36.550} C_DIS
   LIN {X -4.379, Y -26.568, Z 36.550} C_DIS
   LIN {X -4.695, Y -26.349, Z 36.550} C_DIS
   LIN {X -6.080, Y -25.396, Z 36.550}
   LaserEnd_Ext()
   LIN {X -1.938, Y 13.186, Z 36.550}
   LaserStart_Ext()
   LIN {X -1.942, Y 12.606, Z 36.550} C_DIS
   LIN {X -2.081, Y 11.393, Z 36.550} C_DIS
   LIN {X -2.833, Y 4.478, Z 36.550} C_DIS
   LIN {X -4.003, Y -0.912, Z 36.550} C_DIS
   LIN {X -4.331, Y -2.396, Z 36.550} C_DIS
   LIN {X -4.630, Y -3.372, Z 36.550} C_DIS
   LIN {X -5.795, Y -7.180, Z 36.550} C_DIS
   LIN {X -6.432, Y -8.871, Z 36.550} C_DIS
   LIN {X -7.225, Y -10.988, Z 36.550} C_DIS
   LIN {X -7.858, Y -12.446, Z 36.550} C_DIS
   LIN {X -8.801, Y -14.580, Z 36.550} C_DIS
   LIN {X -9.744, Y -16.444, Z 36.550} C_DIS
   LIN {X -10.390, Y -17.742, Z 36.550} C_DIS
   LIN {X -10.792, Y -18.998, Z 36.550} C_DIS
   LIN {X -11.369, Y -20.758, Z 36.550} C_DIS
   LIN {X -11.115, Y -24.424, Z 36.550} C_DIS
   LIN {X -9.352, Y -27.770, Z 36.550} C_DIS
   LIN {X -7.495, Y -29.287, Z 36.550} C_DIS
   LIN {X -6.827, Y -29.839, Z 36.550} C_DIS
   LIN {X -3.815, Y -30.852, Z 36.550} C_DIS
   LIN {X -1.510, Y -30.839, Z 36.550} C_DIS
   LIN {X -1.110, Y -30.843, Z 36.550} C_DIS
   LIN {X -0.511, Y -30.618, Z 36.550} C_DIS
   LIN {X 2.449, Y -29.476, Z 36.550} C_DIS
   LIN {X 4.430, Y -27.490, Z 36.550} C_DIS
   LIN {X 5.138, Y -26.769, Z 36.550} C_DIS
   LIN {X 5.623, Y -25.633, Z 36.550} C_DIS
   LIN {X 6.324, Y -24.010, Z 36.550} C_DIS
   LIN {X 6.591, Y -22.849, Z 36.550} C_DIS
   LIN {X 7.044, Y -20.828, Z 36.550} C_DIS
   LIN {X 7.612, Y -17.954, Z 36.550} C_DIS
   LIN {X 8.253, Y -14.087, Z 36.550} C_DIS
   LIN {X 8.604, Y -11.347, Z 36.550} C_DIS
   LIN {X 8.838, Y -9.432, Z 36.550} C_DIS
   LIN {X 9.077, Y -6.340, Z 36.550} C_DIS
   LIN {X 9.274, Y -3.917, Z 36.550} C_DIS
   LIN {X 9.325, Y -1.546, Z 36.550} C_DIS
   LIN {X 9.410, Y 4.298, Z 36.550} C_DIS
   LIN {X 9.244, Y 7.246, Z 36.550} C_DIS
   LIN {X 9.054, Y 11.249, Z 36.550} C_DIS
   LIN {X 8.915, Y 12.583, Z 36.550} C_DIS
   LIN {X 7.836, Y 20.343, Z 36.550} C_DIS
   LIN {X 7.492, Y 22.616, Z 36.550} C_DIS
   LIN {X 6.715, Y 26.187, Z 36.550} C_DIS
   LIN {X 6.221, Y 28.414, Z 36.550} C_DIS
   LIN {X 5.142, Y 32.464, Z 36.550} C_DIS
   LIN {X 5.102, Y 32.599, Z 36.550} C_DIS
   LIN {X 4.201, Y 35.578, Z 36.550} C_DIS
   LIN {X 3.895, Y 36.509, Z 36.550} C_DIS
   LIN {X 3.458, Y 37.828, Z 36.550} C_DIS
   LIN {X 2.929, Y 39.329, Z 36.550} C_DIS
   LIN {X 2.829, Y 39.615, Z 36.550} C_DIS
   LIN {X 2.762, Y 39.798, Z 36.550} C_DIS
   LIN {X 2.314, Y 41.012, Z 36.550} C_DIS
   LIN {X 1.674, Y 42.074, Z 36.550} C_DIS
   LIN {X 1.554, Y 42.272, Z 36.550} C_DIS
   LIN {X 1.253, Y 42.489, Z 36.550} C_DIS
   LIN {X 0.143, Y 43.293, Z 36.550} C_DIS
   LIN {X -0.719, Y 43.458, Z 36.550} C_DIS
   LIN {X -1.572, Y 43.619, Z 36.550} C_DIS
   LIN {X -3.351, Y 42.955, Z 36.550} C_DIS
   LIN {X -3.974, Y 42.707, Z 36.550} C_DIS
   LIN {X -4.445, Y 42.120, Z 36.550} C_DIS
   LIN {X -4.970, Y 41.471, Z 36.550} C_DIS
   LIN {X -5.310, Y 40.186, Z 36.550} C_DIS
   LIN {X -5.407, Y 39.829, Z 36.550} C_DIS
   LIN {X -5.375, Y 39.588, Z 36.550} C_DIS
   LIN {X -5.218, Y 38.440, Z 36.550} C_DIS
   LIN {X -4.859, Y 37.242, Z 36.550} C_DIS
   LIN {X -4.421, Y 35.703, Z 36.550} C_DIS
   LIN {X -4.029, Y 34.174, Z 36.550} C_DIS
   LIN {X -3.834, Y 33.405, Z 36.550} C_DIS
   LIN {X -3.515, Y 31.930, Z 36.550} C_DIS
   LIN {X -3.219, Y 30.575, Z 36.550} C_DIS
   LIN {X -3.056, Y 29.647, Z 36.550} C_DIS
   LIN {X -2.652, Y 27.296, Z 36.550} C_DIS
   LIN {X -2.057, Y 21.711, Z 36.550} C_DIS
   LIN {X -2.026, Y 21.410, Z 36.550} C_DIS
   LIN {X -2.012, Y 21.274, Z 36.550} C_DIS
   LIN {X -1.976, Y 20.887, Z 36.550} C_DIS
   LIN {X -1.938, Y 13.186, Z 36.550}
   LaserEnd_Ext()
   LIN {X -10.280, Y -20.644, Z 36.550}
   LaserStart_Ext()
   LIN {X -10.280, Y -22.011, Z 36.550}
   LaserEnd_Ext()
   LIN {X -9.280, Y -25.777, Z 36.550}
   LaserStart_Ext()
   LIN {X -9.280, Y -17.755, Z 36.550}
   LaserEnd_Ext()
   LIN {X -8.280, Y -15.764, Z 36.550}
   LaserStart_Ext()
   LIN {X -8.280, Y -20.983, Z 36.550}
   LaserEnd_Ext()
   LIN {X -8.280, Y -22.784, Z 36.550}
   LaserStart_Ext()
   LIN {X -8.280, Y -27.355, Z 36.550}
   LaserEnd_Ext()
   LIN {X -7.280, Y -28.172, Z 36.550}
   LaserStart_Ext()
   LIN {X -7.280, Y -25.354, Z 36.550}
   LaserEnd_Ext()
   LIN {X -7.280, Y -18.451, Z 36.550}
   LaserStart_Ext()
   LIN {X -7.280, Y -13.611, Z 36.550}
   LaserEnd_Ext()
   LIN {X -6.280, Y -11.317, Z 36.550}
   LaserStart_Ext()
   LIN {X -6.280, Y -17.500, Z 36.550}
   LaserEnd_Ext()
   LIN {X -6.280, Y -26.472, Z 36.550}
   LaserStart_Ext()
   LIN {X -6.280, Y -28.968, Z 36.550}
   LaserEnd_Ext()
   LIN {X -5.280, Y -29.304, Z 36.550}
   LaserStart_Ext()
   LIN {X -5.280, Y -27.160, Z 36.550}
   LaserEnd_Ext()
   LIN {X -5.280, Y -16.668, Z 36.550}
   LaserStart_Ext()
   LIN {X -5.280, Y -8.650, Z 36.550}
   LaserEnd_Ext()
   LIN {X -4.280, Y 40.170, Z 36.550}
   LaserStart_Ext()
   LIN {X -4.280, Y 38.960, Z 36.550}
   LaserEnd_Ext()
   LIN {X -4.280, Y -5.646, Z 36.550}
   LaserStart_Ext()
   LIN {X -4.280, Y -16.354, Z 36.550}
   LaserEnd_Ext()
   LIN {X -4.280, Y -27.604, Z 36.550}
   LaserStart_Ext()
   LIN {X -4.280, Y -29.640, Z 36.550}
   LaserEnd_Ext()
   LIN {X -3.280, Y -29.849, Z 36.550}
   LaserStart_Ext()
   LIN {X -3.280, Y -27.787, Z 36.550}
   LaserEnd_Ext()
   LIN {X -3.280, Y -16.084, Z 36.550}
   LaserStart_Ext()
   LIN {X -3.280, Y -2.274, Z 36.550}
   LaserEnd_Ext()
   LIN {X -3.280, Y 35.279, Z 36.550}
   LaserStart_Ext()
   LIN {X -3.280, Y 41.907, Z 36.550}
   LaserEnd_Ext()
   LIN {X -2.280, Y 42.288, Z 36.550}
   LaserStart_Ext()
   LIN {X -2.280, Y 30.962, Z 36.550}
   LaserEnd_Ext()
   LIN {X -2.280, Y 2.314, Z 36.550}
   LaserStart_Ext()
   LIN {X -2.280, Y -15.977, Z 36.550}
   LaserEnd_Ext()
   LIN {X -2.280, Y -27.933, Z 36.550}
   LaserStart_Ext()
   LIN {X -2.280, Y -29.843, Z 36.550}
   LaserEnd_Ext()
   LIN {X -1.280, Y -29.838, Z 36.550}
   LaserStart_Ext()
   LIN {X -1.280, Y -27.703, Z 36.550}
   LaserEnd_Ext()
   LIN {X -1.280, Y -16.153, Z 36.550}
   LaserStart_Ext()
   LIN {X -1.280, Y 9.513, Z 36.550}
   LaserEnd_Ext()
   LIN {X -1.280, Y 23.855, Z 36.550}
   LaserStart_Ext()
   LIN {X -1.280, Y 42.546, Z 36.550}
   LaserEnd_Ext()
   LIN {X -0.280, Y 42.356, Z 36.550}
   LaserStart_Ext()
   LIN {X -0.280, Y -16.333, Z 36.550}
   LaserEnd_Ext()
   LIN {X -0.280, Y -27.458, Z 36.550}
   LaserStart_Ext()
   LIN {X -0.280, Y -29.457, Z 36.550}
   LaserEnd_Ext()
   LIN {X 0.720, Y -29.071, Z 36.550}
   LaserStart_Ext()
   LIN {X 0.720, Y -26.937, Z 36.550}
   LaserEnd_Ext()
   LIN {X 0.720, Y -16.942, Z 36.550}
   LaserStart_Ext()
   LIN {X 0.720, Y 41.641, Z 36.550}
   LaserEnd_Ext()
   LIN {X 1.720, Y 39.734, Z 36.550}
   LaserStart_Ext()
   LIN {X 1.720, Y -17.638, Z 36.550}
   LaserEnd_Ext()
   LIN {X 1.720, Y -26.144, Z 36.550}
   LaserStart_Ext()
   LIN {X 1.720, Y -28.686, Z 36.550}
   LaserEnd_Ext()
   LIN {X 2.720, Y -27.789, Z 36.550}
   LaserStart_Ext()
   LIN {X 2.720, Y -24.684, Z 36.550}
   LaserEnd_Ext()
   LIN {X 2.720, Y -19.175, Z 36.550}
   LaserStart_Ext()
   LIN {X 2.720, Y 36.875, Z 36.550}
   LaserEnd_Ext()
   LIN {X 3.720, Y 33.713, Z 36.550}
   LaserStart_Ext()
   LIN {X 3.720, Y -26.786, Z 36.550}
   LaserEnd_Ext()
   LIN {X 4.720, Y -25.201, Z 36.550}
   LaserStart_Ext()
   LIN {X 4.720, Y 30.164, Z 36.550}
   LaserEnd_Ext()
   LIN {X 5.720, Y 26.053, Z 36.550}
   LaserStart_Ext()
   LIN {X 5.720, Y -22.163, Z 36.550}
   LaserEnd_Ext()
   LIN {X 6.720, Y -17.222, Z 36.550}
   LaserStart_Ext()
   LIN {X 6.720, Y 21.035, Z 36.550}
   LaserEnd_Ext()
   LIN {X 7.720, Y 13.918, Z 36.550}
   LaserStart_Ext()
   LIN {X 7.720, Y -10.339, Z 36.550}
   LaserEnd_Ext()
   LIN {X -6.713, Y -24.190, Z 37.400}
   LaserStart_Ext()
   LIN {X -7.089, Y -23.583, Z 37.400} C_DIS
   LIN {X -7.184, Y -22.844, Z 37.400} C_DIS
   LIN {X -7.352, Y -21.513, Z 37.400} C_DIS
   LIN {X -6.768, Y -20.010, Z 37.400} C_DIS
   LIN {X -6.347, Y -18.887, Z 37.400} C_DIS
   LIN {X -5.750, Y -18.344, Z 37.400} C_DIS
   LIN {X -4.792, Y -17.531, Z 37.400} C_DIS
   LIN {X -3.611, Y -17.212, Z 37.400} C_DIS
   LIN {X -2.518, Y -16.891, Z 37.400} C_DIS
   LIN {X -1.214, Y -17.116, Z 37.400} C_DIS
   LIN {X -0.446, Y -17.251, Z 37.400} C_DIS
   LIN {X 0.078, Y -17.615, Z 37.400} C_DIS
   LIN {X 1.301, Y -18.460, Z 37.400} C_DIS
   LIN {X 2.216, Y -20.154, Z 37.400} C_DIS
   LIN {X 2.507, Y -20.699, Z 37.400} C_DIS
   LIN {X 2.514, Y -21.297, Z 37.400} C_DIS
   LIN {X 2.537, Y -22.875, Z 37.400} C_DIS
   LIN {X 1.579, Y -24.855, Z 37.400} C_DIS
   LIN {X 1.475, Y -25.072, Z 37.400} C_DIS
   LIN {X 1.268, Y -25.238, Z 37.400} C_DIS
   LIN {X -0.147, Y -26.363, Z 37.400} C_DIS
   LIN {X -1.746, Y -26.760, Z 37.400} C_DIS
   LIN {X -2.278, Y -26.890, Z 37.400} C_DIS
   LIN {X -2.997, Y -26.758, Z 37.400} C_DIS
   LIN {X -4.292, Y -26.524, Z 37.400} C_DIS
   LIN {X -5.103, Y -25.970, Z 37.400} C_DIS
   LIN {X -5.995, Y -25.356, Z 37.400} C_DIS
   LIN {X -6.713, Y -24.190, Z 37.400}
   LaserEnd_Ext()
   LIN {X 9.424, Y 4.383, Z 37.400}
   LaserStart_Ext()
   LIN {X 9.179, Y 8.737, Z 37.400} C_DIS
   LIN {X 9.066, Y 11.133, Z 37.400} C_DIS
   LIN {X 8.982, Y 11.931, Z 37.400} C_DIS
   LIN {X 7.681, Y 21.293, Z 37.400} C_DIS
   LIN {X 7.500, Y 22.485, Z 37.400} C_DIS
   LIN {X 7.092, Y 24.357, Z 37.400} C_DIS
   LIN {X 6.169, Y 28.520, Z 37.400} C_DIS
   LIN {X 5.416, Y 31.351, Z 37.400} C_DIS
   LIN {X 5.070, Y 32.603, Z 37.400} C_DIS
   LIN {X 4.272, Y 35.227, Z 37.400} C_DIS
   LIN {X 4.081, Y 35.826, Z 37.400} C_DIS
   LIN {X 3.699, Y 36.969, Z 37.400} C_DIS
   LIN {X 3.399, Y 37.876, Z 37.400} C_DIS
   LIN {X 3.220, Y 38.383, Z 37.400} C_DIS
   LIN {X 2.760, Y 39.679, Z 37.400} C_DIS
   LIN {X 2.273, Y 40.992, Z 37.400} C_DIS
   LIN {X 2.187, Y 41.163, Z 37.400} C_DIS
   LIN {X 1.480, Y 42.330, Z 37.400} C_DIS
   LIN {X 0.479, Y 43.051, Z 37.400} C_DIS
   LIN {X 0.067, Y 43.347, Z 37.400} C_DIS
   LIN {X -0.626, Y 43.476, Z 37.400} C_DIS
   LIN {X -1.650, Y 43.669, Z 37.400} C_DIS
   LIN {X -2.259, Y 43.442, Z 37.400} C_DIS
   LIN {X -4.097, Y 42.709, Z 37.400} C_DIS
   LIN {X -4.767, Y 41.874, Z 37.400} C_DIS
   LIN {X -5.070, Y 41.448, Z 37.400} C_DIS
   LIN {X -5.218, Y 40.859, Z 37.400} C_DIS
   LIN {X -5.473, Y 39.921, Z 37.400} C_DIS
   LIN {X -5.341, Y 38.924, Z 37.400} C_DIS
   LIN {X -5.284, Y 38.482, Z 37.400} C_DIS
   LIN {X -5.210, Y 38.242, Z 37.400} C_DIS
   LIN {X -4.921, Y 37.284, Z 37.400} C_DIS
   LIN {X -4.583, Y 36.110, Z 37.400} C_DIS
   LIN {X -4.480, Y 35.746, Z 37.400} C_DIS
   LIN {X -4.282, Y 34.975, Z 37.400} C_DIS
   LIN {X -3.888, Y 33.450, Z 37.400} C_DIS
   LIN {X -3.568, Y 32.004, Z 37.400} C_DIS
   LIN {X -3.266, Y 30.622, Z 37.400} C_DIS
   LIN {X -2.819, Y 28.080, Z 37.400} C_DIS
   LIN {X -2.708, Y 27.461, Z 37.400} C_DIS
   LIN {X -2.140, Y 22.141, Z 37.400} C_DIS
   LIN {X -2.079, Y 21.572, Z 37.400} C_DIS
   LIN {X -2.055, Y 21.345, Z 37.400} C_DIS
   LIN {X -2.007, Y 20.970, Z 37.400} C_DIS
   LIN {X -1.965, Y 12.991, Z 37.400} C_DIS
   LIN {X -1.950, Y 12.605, Z 37.400} C_DIS
   LIN {X -2.056, Y 11.600, Z 37.400} C_DIS
   LIN {X -2.837, Y 4.422, Z 37.400} C_DIS
   LIN {X -4.321, Y -2.416, Z 37.400} C_DIS
   LIN {X -5.799, Y -7.270, Z 37.400} C_DIS
   LIN {X -5.908, Y -7.572, Z 37.400} C_DIS
   LIN {X -7.163, Y -10.923, Z 37.400} C_DIS
   LIN {X -8.352, Y -13.658, Z 37.400} C_DIS
   LIN {X -8.771, Y -14.607, Z 37.400} C_DIS
   LIN {X -9.191, Y -15.436, Z 37.400} C_DIS
   LIN {X -10.324, Y -17.713, Z 37.400} C_DIS
   LIN {X -11.029, Y -19.916, Z 37.400} C_DIS
   LIN {X -11.296, Y -20.731, Z 37.400} C_DIS
   LIN {X -11.175, Y -22.476, Z 37.400} C_DIS
   LIN {X -11.030, Y -24.432, Z 37.400} C_DIS
   LIN {X -10.356, Y -25.681, Z 37.400} C_DIS
   LIN {X -9.262, Y -27.738, Z 37.400} C_DIS
   LIN {X -8.123, Y -28.669, Z 37.400} C_DIS
   LIN {X -6.795, Y -29.765, Z 37.400} C_DIS
   LIN {X -3.682, Y -30.812, Z 37.400} C_DIS
   LIN {X -1.950, Y -30.803, Z 37.400} C_DIS
   LIN {X -0.929, Y -30.775, Z 37.400} C_DIS
   LIN {X 0.353, Y -30.259, Z 37.400} C_DIS
   LIN {X 2.550, Y -29.413, Z 37.400} C_DIS
   LIN {X 3.498, Y -28.462, Z 37.400} C_DIS
   LIN {X 5.230, Y -26.696, Z 37.400} C_DIS
   LIN {X 6.398, Y -23.959, Z 37.400} C_DIS
   LIN {X 7.118, Y -20.757, Z 37.400} C_DIS
   LIN {X 7.443, Y -19.109, Z 37.400} C_DIS
   LIN {X 7.685, Y -17.852, Z 37.400} C_DIS
   LIN {X 8.088, Y -15.357, Z 37.400} C_DIS
   LIN {X 8.311, Y -14.013, Z 37.400} C_DIS
   LIN {X 8.436, Y -13.039, Z 37.400} C_DIS
   LIN {X 8.884, Y -9.375, Z 37.400} C_DIS
   LIN {X 9.286, Y -4.156, Z 37.400} C_DIS
   LIN {X 9.307, Y -3.855, Z 37.400} C_DIS
   LIN {X 9.307, Y -3.671, Z 37.400} C_DIS
   LIN {X 9.424, Y 4.383, Z 37.400}
   LaserEnd_Ext()
   LIN {X -4.862, Y -29.360, Z 37.400}
   LaserStart_Ext()
   LIN {X -0.091, Y -29.360, Z 37.400}
   LaserEnd_Ext()
   LIN {X 2.187, Y -28.360, Z 37.400}
   LaserStart_Ext()
   LIN {X -6.926, Y -28.360, Z 37.400}
   LaserEnd_Ext()
   LIN {X -8.145, Y -27.360, Z 37.400}
   LaserStart_Ext()
   LIN {X -4.839, Y -27.360, Z 37.400}
   LaserEnd_Ext()
   LIN {X -0.012, Y -27.360, Z 37.400}
   LaserStart_Ext()
   LIN {X 3.178, Y -27.360, Z 37.400}
   LaserEnd_Ext()
   LIN {X 4.159, Y -26.360, Z 37.400}
   LaserStart_Ext()
   LIN {X 1.464, Y -26.360, Z 37.400}
   LaserEnd_Ext()
   LIN {X -6.300, Y -26.360, Z 37.400}
   LaserStart_Ext()
   LIN {X -8.863, Y -26.360, Z 37.400}
   LaserEnd_Ext()
   LIN {X -9.394, Y -25.360, Z 37.400}
   LaserStart_Ext()
   LIN {X -7.167, Y -25.360, Z 37.400}
   LaserEnd_Ext()
   LIN {X 2.446, Y -25.360, Z 37.400}
   LaserStart_Ext()
   LIN {X 4.713, Y -25.360, Z 37.400}
   LaserEnd_Ext()
   LIN {X 5.139, Y -24.360, Z 37.400}
   LaserStart_Ext()
   LIN {X 2.929, Y -24.360, Z 37.400}
   LaserEnd_Ext()
   LIN {X -7.784, Y -24.360, Z 37.400}
   LaserStart_Ext()
   LIN {X -9.933, Y -24.360, Z 37.400}
   LaserEnd_Ext()
   LIN {X -10.107, Y -23.360, Z 37.400}
   LaserStart_Ext()
   LIN {X -8.126, Y -23.360, Z 37.400}
   LaserEnd_Ext()
   LIN {X 3.413, Y -23.360, Z 37.400}
   LaserStart_Ext()
   LIN {X 5.510, Y -23.360, Z 37.400}
   LaserEnd_Ext()
   LIN {X 5.734, Y -22.360, Z 37.400}
   LaserStart_Ext()
   LIN {X 3.530, Y -22.360, Z 37.400}
   LaserEnd_Ext()
   LIN {X -8.253, Y -22.360, Z 37.400}
   LaserStart_Ext()
   LIN {X -10.180, Y -22.360, Z 37.400}
   LaserEnd_Ext()
   LIN {X -10.250, Y -21.360, Z 37.400}
   LaserStart_Ext()
   LIN {X -8.340, Y -21.360, Z 37.400}
   LaserEnd_Ext()
   LIN {X 3.515, Y -21.360, Z 37.400}
   LaserStart_Ext()
   LIN {X 5.958, Y -21.360, Z 37.400}
   LaserEnd_Ext()
   LIN {X 6.177, Y -20.360, Z 37.400}
   LaserStart_Ext()
   LIN {X 3.447, Y -20.360, Z 37.400}
   LaserEnd_Ext()
   LIN {X -7.977, Y -20.360, Z 37.400}
   LaserStart_Ext()
   LIN {X -10.122, Y -20.360, Z 37.400}
   LaserEnd_Ext()
   LIN {X -9.801, Y -19.360, Z 37.400}
   LaserStart_Ext()
   LIN {X -7.592, Y -19.360, Z 37.400}
   LaserEnd_Ext()
   LIN {X 2.923, Y -19.360, Z 37.400}
   LaserStart_Ext()
   LIN {X 6.374, Y -19.360, Z 37.400}
   LaserEnd_Ext()
   LIN {X 6.569, Y -18.360, Z 37.400}
   LaserStart_Ext()
   LIN {X 2.384, Y -18.360, Z 37.400}
   LaserEnd_Ext()
   LIN {X -7.196, Y -18.360, Z 37.400}
   LaserStart_Ext()
   LIN {X -9.481, Y -18.360, Z 37.400}
   LaserEnd_Ext()
   LIN {X -9.031, Y -17.360, Z 37.400}
   LaserStart_Ext()
   LIN {X -6.136, Y -17.360, Z 37.400}
   LaserEnd_Ext()
   LIN {X 1.469, Y -17.360, Z 37.400}
   LaserStart_Ext()
   LIN {X 6.751, Y -17.360, Z 37.400}
   LaserEnd_Ext()
   LIN {X 6.913, Y -16.360, Z 37.400}
   LaserStart_Ext()
   LIN {X 0.006, Y -16.360, Z 37.400}
   LaserEnd_Ext()
   LIN {X -4.291, Y -16.360, Z 37.400}
   LaserStart_Ext()
   LIN {X -8.534, Y -16.360, Z 37.400}
